# B&R Automation Studio project CombinedLinenCleanA6
Automation Studio 4.10.2.37; technology packages: mappView 5.17.0

## Configuration CP1584

CPU 5APC2200.AL14-000, AutomationRuntime B4.63, Build 4.1.2, Safety 0.0, Vc V4.72.3

### Task classes (Cpu.sw)
```
Cyclic#2 (cycle 10000 us, tolerance 10000 us):
  zzstd <- Sequences.zzstd.prg
  zztc2str <- Sequences.zztc2str.prg
  zzforcei <- Sequences.zzforcei.prg
  zzconst <- Sequences.zzconst.prg
  zztrip <- Sequences.zztrip.prg
  zzbagsfl <- Sequences.zzbagsfl.prg
  zzbitcal <- Sequences.zzbitcal.prg
  zcusfifo <- Sequences.zcusfifo.prg
  zzStnSer <- Sequences.10ms.zzStnSer.prg
  1_clu_1 <- Sequences.10ms.1_clu_1.prg
  2_cvc1 <- Sequences.10ms.2_cvc1.prg
  3_cic1 <- Sequences.10ms.3_cic1.prg
  4_cic2 <- Sequences.10ms.4_cic2.prg
  5_cic3 <- Sequences.10ms.5_cic3.prg
  6_sdc1 <- Sequences.10ms.6_sdc1.prg [disabled]
  7_sdc2 <- Sequences.10ms.7_sdc2.prg
  8_sdc3 <- Sequences.10ms.8_sdc3.prg
  9_sdc4 <- Sequences.10ms.9_sdc4.prg
  10_sdc5 <- Sequences.10ms.10_sdc5.prg
  11_sdc6 <- Sequences.10ms.11_sdc6.prg
  12_ebag <- Sequences.10ms.12_ebag.prg
  13_fb_eb <- Sequences.10ms.13_fb_eb.prg
  14_cvc2 <- Sequences.10ms.14_cvc2.prg
  15_cdc7 <- Sequences.10ms.15_cdc7.prg
  16_cic4 <- Sequences.10ms.16_cic4.prg
  17_cp12 <- Sequences.10ms.17_cp12.prg
  18_cdc8 <- Sequences.10ms.18_cdc8.prg
  19_cp13 <- Sequences.10ms.19_cp13.prg
  20_cpc1 <- Sequences.10ms.20_cpc1.prg
  21_cic6 <- Sequences.10ms.21_cic6.prg
  22_cic7 <- Sequences.10ms.22_cic7.prg
  23_Ebag <- Sequences.10ms.23_Ebag.prg
  24_csb1 <- Sequences.10ms.24_csb1.prg
  25_cp16 <- Sequences.10ms.25_cp16.prg
  26_cic8 <- Sequences.10ms.26_cic8.prg
  27_csb2 <- Sequences.10ms.27_csb2.prg
  ssr <- Sequences.10ms.ssr.prg
  can_live <- Sequences.can_live.prg
  zzio <- Sequences.zzio.prg
  zztcpip <- Sequences.zztcpip.prg
  zzuld_3 <- Sequences.zzuld_3.prg
  zzreport <- Sequences.zzreport.prg
  zztc2end <- Sequences.zztc2end.prg
Cyclic#5:
  zzweigh <- zzweigh.prg [disabled]
  can_drv2 <- Mewa.200ms.CAN.can_drv2.prg
  zzstn_q <- Sequences.zzstn_q.prg
  zzalarms <- Sequences.zzalarms.prg
  zztime <- zztime.prg
  zztc2end1 <- zztc2end.prg
DataObjects: can_cmd <- Mewa.200ms.CAN.can_cmd.dob
Binaries: TCData, udbdef, mvLoader, sysconf, ashwd, asfw, arconfig, iomap, ashwac
Libraries: DataBackUp, AsDb, standard, runtime, FileIO, Ethernet, dvframe, DataObj, OPERATOR, CAN_Lib, AsTime, AsString, SupLib4, sys_lib, AsTCP, KGstring, Visapi, AsETH, AsBrStr, AsBrWStr, AsUSB, AsMem, AsArLog, AsUDP, brsystem, AsIODiag, AsARCfg, AsIecCon, IecCheck, arssl, zzSQL_Lib
```

### Hardware
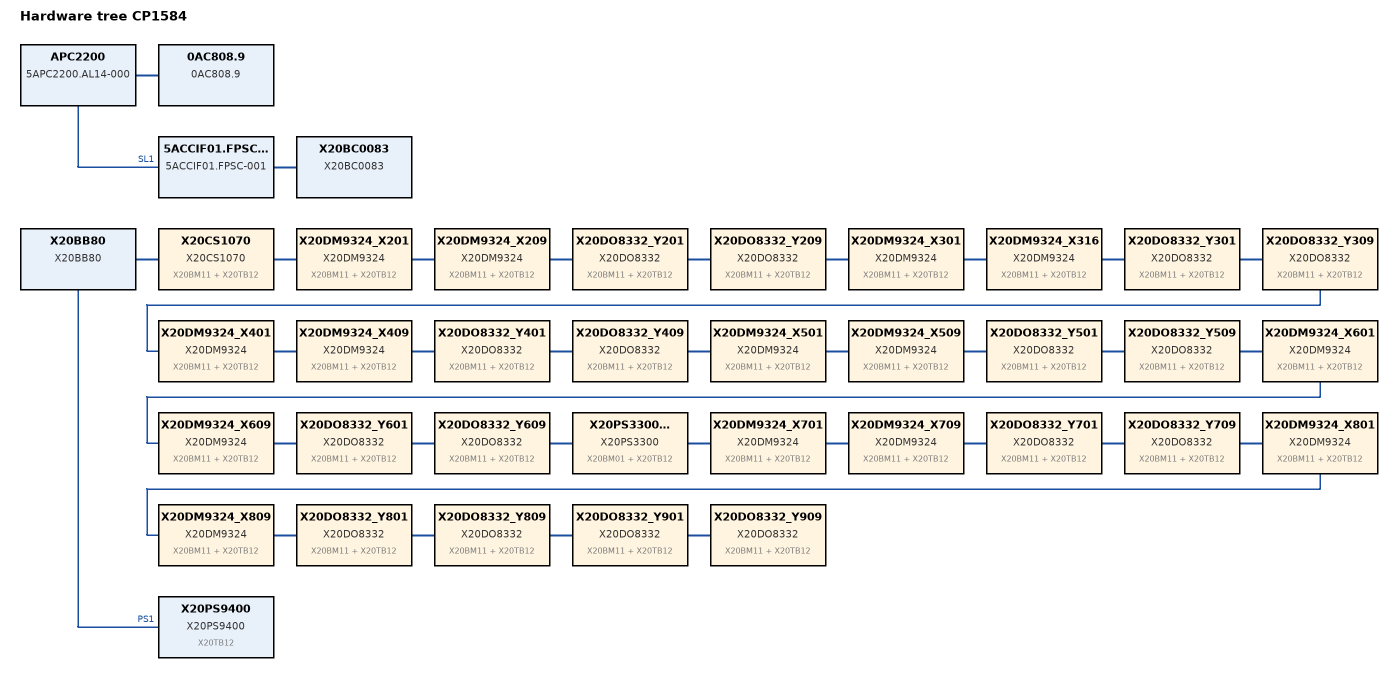
```
0AC808.9 : 0AC808.9 v1.0.0.0  [ETH1 -> APC2200.IF3 [Cable Type=PowerlinkCable, Length=10, Version=1.0.0.3]]
5ACCIF01.FPSC-001 : 5ACCIF01.FPSC-001 v1.9.1.0  [SL -> APC2200.SL1]
APC2200 : 5APC2200.AL14-000 v2.0.3.0
  Connector IF3:
    AssignedOperatingSystem = ARemb
    ActivateDevice = 1
    Baudrate = 100
    InaNodeNumber = 21
    ActivateANSL = 0
  Connector IF4:
    AssignedOperatingSystem = ARemb
    ActivateDevice = 1
    Mode = Manual
    InternetAddress = 10.8.4.21
    SubnetMask = 255.255.240.0
  Connector IF5:
    AssignedOperatingSystem = ARemb
  Connector IF6:
    AssignedOperatingSystem = ARemb
  ConfigurationID = AS4_2_BaseStandard_Supertrack
  UserRamDevice = PCI.1.PPC21xx.SRAM
  UserRamSize = 200000
  RemMemDevice = PCI.1.PPC21xx.SRAM
  RemMemSize = 200000
  PermanentPvSize = 46756
  RemanentGlobalPvSize = 8944
  VolatileGlobalPvSize = 450000
  EnableUsbRemoteInstall = 1
  EnableCfRemoteInstall = 1
  RebootPowerfail = 2
  Cyclic1Duration = 1000
  Cyclic1Tolerance = 1000
  Cyclic2Duration = 10000
  Cyclic2Tolerance = 10000
  FileDevice1
  FileDeviceName1 = USBStick
  FileDevicePath1 = /bd0\
  FileDevice2
  FileDeviceName2 = UserPart
  FileDevicePath2 = F:\
  EthernetHostName = SupertrackPLC
  EthernetDefaultGateway = 10.8.15.254
  FtpUser1
  FtpUsername1 = admin
  FtpUserPassword1 = vwQCGOhDKwuFhUdMhisKVJgiKzmoNTQazzJQnTTJsZU=  // admin
  FtpUserSalt1 = XFuy8Eo/
  FTPAccessRight1 = 0
  ActivateOpcUa = 1
  OpcUaInformationModels_PV_Version = 1
X20BB80 : X20BB80 v1.1.0.0
X20BC0083 : X20BC0083 v2.14.0.0  [PLK1 -> 5ACCIF01.FPSC-001.IF1 (NodeNumber=1) [Cable Type=PowerlinkCable, Length=10, Version=1.0.0.3]; SL -> X20BB80.SL1]
  Supervision = off
X20BM01 : X20BM01 v2.1.0.0  [X2X1 -> X20BM11t.X2X2]
X20BM11 : X20BM11 v1.1.0.0  [X2X1 -> X20BB80.IF1]
X20BM11a : X20BM11 v1.1.0.0  [X2X1 -> X20BM11.X2X2]
X20BM11aa : X20BM11 v1.1.0.0  [X2X1 -> X20BM11z.X2X2]
X20BM11ab : X20BM11 v1.1.0.0  [X2X1 -> X20BM11aa.X2X2]
X20BM11ac : X20BM11 v1.1.0.0  [X2X1 -> X20BM11ab.X2X2]
X20BM11ad : X20BM11 v1.1.0.0  [X2X1 -> X20BM11ac.X2X2]
X20BM11b : X20BM11 v1.1.0.0  [X2X1 -> X20BM11a.X2X2]
X20BM11c : X20BM11 v1.1.0.0  [X2X1 -> X20BM11b.X2X2]
X20BM11d : X20BM11 v1.1.0.0  [X2X1 -> X20BM11e.X2X2]
X20BM11e : X20BM11 v1.1.0.0  [X2X1 -> X20BM11c.X2X2]
X20BM11f : X20BM11 v1.1.0.0  [X2X1 -> X20BM11d.X2X2]
X20BM11g : X20BM11 v1.1.0.0  [X2X1 -> X20BM11s.X2X2]
X20BM11h : X20BM11 v1.1.0.0  [X2X1 -> X20BM11f.X2X2]
X20BM11i : X20BM11 v1.1.0.0  [X2X1 -> X20BM11h.X2X2]
X20BM11j : X20BM11 v1.1.0.0  [X2X1 -> X20BM11i.X2X2]
X20BM11k : X20BM11 v1.1.0.0  [X2X1 -> X20BM11j.X2X2]
X20BM11l : X20BM11 v1.1.0.0  [X2X1 -> X20BM11k.X2X2]
X20BM11m : X20BM11 v1.1.0.0  [X2X1 -> X20BM11l.X2X2]
X20BM11n : X20BM11 v1.1.0.0  [X2X1 -> X20BM11m.X2X2]
X20BM11o : X20BM11 v1.1.0.0  [X2X1 -> X20BM11n.X2X2]
X20BM11p : X20BM11 v1.1.0.0  [X2X1 -> X20BM11o.X2X2]
X20BM11q : X20BM11 v1.1.0.0  [X2X1 -> X20BM11p.X2X2]
X20BM11r : X20BM11 v1.1.0.0  [X2X1 -> X20BM11q.X2X2]
X20BM11s : X20BM11 v1.1.0.0  [X2X1 -> X20BM11r.X2X2]
X20BM11t : X20BM11 v1.1.0.0  [X2X1 -> X20BM11g.X2X2]
X20BM11u : X20BM11 v1.1.0.0  [X2X1 -> X20BM01.X2X2]
X20BM11v : X20BM11 v1.1.0.0  [X2X1 -> X20BM11u.X2X2]
X20BM11w : X20BM11 v1.1.0.0  [X2X1 -> X20BM11v.X2X2]
X20BM11x : X20BM11 v1.1.0.0  [X2X1 -> X20BM11w.X2X2]
X20BM11y : X20BM11 v1.1.0.0  [X2X1 -> X20BM11x.X2X2]
X20BM11z : X20BM11 v1.1.0.0  [X2X1 -> X20BM11y.X2X2]
X20CS1070 : X20CS1070 v1.8.0.0  [SS1 -> X20TB12af.SS; SL -> X20BM11.SL1]
  FunctionModel = Stream1xCan
  Supervision = off
X20DM9324_X201 : X20DM9324 v1.2.0.0  [SS1 -> X20TB12a.SS; SL -> X20BM11a.SL1]
  Supervision = off
X20DM9324_X209 : X20DM9324 v1.2.0.0  [SS1 -> X20TB12b.SS; SL -> X20BM11b.SL1]
  Supervision = off
X20DM9324_X301 : X20DM9324 v1.2.0.0  [SS1 -> X20TB12d.SS; SL -> X20BM11d.SL1]
  Supervision = off
X20DM9324_X316 : X20DM9324 v1.2.0.0  [SS1 -> X20TB12f.SS; SL -> X20BM11f.SL1]
  Supervision = off
X20DM9324_X401 : X20DM9324 v1.2.0.0  [SS1 -> X20TB12j.SS; SL -> X20BM11j.SL1]
  Supervision = off
X20DM9324_X409 : X20DM9324 v1.2.0.0  [SS1 -> X20TB12k.SS; SL -> X20BM11k.SL1]
  Supervision = off
X20DM9324_X501 : X20DM9324 v1.2.0.0  [SS1 -> X20TB12n.SS; SL -> X20BM11n.SL1]
  Supervision = off
X20DM9324_X509 : X20DM9324 v1.2.0.0  [SS1 -> X20TB12o.SS; SL -> X20BM11o.SL1]
  Supervision = off
X20DM9324_X601 : X20DM9324 v1.2.0.0  [SS1 -> X20TB12r.SS; SL -> X20BM11r.SL1]
  Supervision = off
X20DM9324_X609 : X20DM9324 v1.2.0.0  [SS1 -> X20TB12s.SS; SL -> X20BM11s.SL1]
  Supervision = off
X20DM9324_X701 : X20DM9324 v1.2.0.0  [SS1 -> X20TB12u.SS; SL -> X20BM11u.SL1]
  Supervision = off
X20DM9324_X709 : X20DM9324 v1.2.0.0  [SS1 -> X20TB12v.SS; SL -> X20BM11v.SL1]
  Supervision = off
X20DM9324_X801 : X20DM9324 v1.2.0.0  [SS1 -> X20TB12z.SS; SL -> X20BM11y.SL1]
  Supervision = off
X20DM9324_X809 : X20DM9324 v1.2.0.0  [SS1 -> X20TB12aa.SS; SL -> X20BM11z.SL1]
  Supervision = off
X20DO8332_Y201 : X20DO8332 v1.5.0.0  [SS1 -> X20TB12c.SS; SL -> X20BM11c.SL1]
  Supervision = off
X20DO8332_Y209 : X20DO8332 v1.5.0.0  [SS1 -> X20TB12e.SS; SL -> X20BM11e.SL1]
  Supervision = off
X20DO8332_Y301 : X20DO8332 v1.5.0.0  [SS1 -> X20TB12h.SS; SL -> X20BM11h.SL1]
  Supervision = off
X20DO8332_Y309 : X20DO8332 v1.5.0.0  [SS1 -> X20TB12i.SS; SL -> X20BM11i.SL1]
  Supervision = off
X20DO8332_Y401 : X20DO8332 v1.5.0.0  [SS1 -> X20TB12l.SS; SL -> X20BM11l.SL1]
  Supervision = off
X20DO8332_Y409 : X20DO8332 v1.5.0.0  [SS1 -> X20TB12m.SS; SL -> X20BM11m.SL1]
  Supervision = off
X20DO8332_Y501 : X20DO8332 v1.5.0.0  [SS1 -> X20TB12p.SS; SL -> X20BM11p.SL1]
  Supervision = off
X20DO8332_Y509 : X20DO8332 v1.5.0.0  [SS1 -> X20TB12q.SS; SL -> X20BM11q.SL1]
  Supervision = off
X20DO8332_Y601 : X20DO8332 v1.5.0.0  [SS1 -> X20TB12g.SS; SL -> X20BM11g.SL1]
  Supervision = off
X20DO8332_Y609 : X20DO8332 v1.5.0.0  [SS1 -> X20TB12t.SS; SL -> X20BM11t.SL1]
  Supervision = off
X20DO8332_Y701 : X20DO8332 v1.5.0.0  [SS1 -> X20TB12x.SS; SL -> X20BM11w.SL1]
  Supervision = off
X20DO8332_Y709 : X20DO8332 v1.5.0.0  [SS1 -> X20TB12y.SS; SL -> X20BM11x.SL1]
  Supervision = off
X20DO8332_Y801 : X20DO8332 v1.5.0.0  [SS1 -> X20TB12ab.SS; SL -> X20BM11aa.SL1]
  Supervision = off
X20DO8332_Y809 : X20DO8332 v1.5.0.0  [SS1 -> X20TB12ac.SS; SL -> X20BM11ab.SL1]
  Supervision = off
X20DO8332_Y901 : X20DO8332 v1.5.0.0  [SS1 -> X20TB12ad.SS; SL -> X20BM11ac.SL1]
  Supervision = off
X20DO8332_Y909 : X20DO8332 v1.5.0.0  [SS1 -> X20TB12ae.SS; SL -> X20BM11ad.SL1]
  Supervision = off
X20PS3300_Power : X20PS3300 v1.3.0.0  [SS1 -> X20TB12w.SS; SL -> X20BM01.SL1]
  Supervision = off
X20PS9400 : X20PS9400 v1.8.0.0  [SS1 -> X20TB12.SS; PS -> X20BB80.PS1]
  Supervision = off
X20TB12 : X20TB12 v1.0.0.0
X20TB12a : X20TB12 v1.0.0.0
X20TB12aa : X20TB12 v1.0.0.0
X20TB12ab : X20TB12 v1.0.0.0
X20TB12ac : X20TB12 v1.0.0.0
X20TB12ad : X20TB12 v1.0.0.0
X20TB12ae : X20TB12 v1.0.0.0
X20TB12af : X20TB12 v1.0.0.0
X20TB12b : X20TB12 v1.0.0.0
X20TB12c : X20TB12 v1.0.0.0
X20TB12d : X20TB12 v1.0.0.0
X20TB12e : X20TB12 v1.0.0.0
X20TB12f : X20TB12 v1.0.0.0
X20TB12g : X20TB12 v1.0.0.0
X20TB12h : X20TB12 v1.0.0.0
X20TB12i : X20TB12 v1.0.0.0
X20TB12j : X20TB12 v1.0.0.0
X20TB12k : X20TB12 v1.0.0.0
X20TB12l : X20TB12 v1.0.0.0
X20TB12m : X20TB12 v1.0.0.0
X20TB12n : X20TB12 v1.0.0.0
X20TB12o : X20TB12 v1.0.0.0
X20TB12p : X20TB12 v1.0.0.0
X20TB12q : X20TB12 v1.0.0.0
X20TB12r : X20TB12 v1.0.0.0
X20TB12s : X20TB12 v1.0.0.0
X20TB12t : X20TB12 v1.0.0.0
X20TB12u : X20TB12 v1.0.0.0
X20TB12v : X20TB12 v1.0.0.0
X20TB12w : X20TB12 v1.0.0.0
X20TB12x : X20TB12 v1.0.0.0
X20TB12y : X20TB12 v1.0.0.0
X20TB12z : X20TB12 v1.0.0.0
```

### IoMap.iom - APC2200/IoMap.iom
```iecst
(********************************************************************
 * COPYRIGHT --
 ********************************************************************
 * File: IoMap.iom
 * Author: Dave
 * Created: November 19, 2010
 ********************************************************************
 * IO mapping file
 ********************************************************************)
VAR_CONFIG
	X[2].X01 AT %IX."X20DM9324_X201".DigitalInput01;
	X[2].X02 AT %IX."X20DM9324_X201".DigitalInput02;
	X[2].X03 AT %IX."X20DM9324_X201".DigitalInput03;
	X[2].X04 AT %IX."X20DM9324_X201".DigitalInput04;
	X[2].X05 AT %IX."X20DM9324_X201".DigitalInput05;
	X[2].X06 AT %IX."X20DM9324_X201".DigitalInput06;
	X[2].X07 AT %IX."X20DM9324_X201".DigitalInput07;
	X[2].X08 AT %IX."X20DM9324_X201".DigitalInput08;
	X[2].X09 AT %IX."X20DM9324_X209".DigitalInput01;
	X[2].X10 AT %IX."X20DM9324_X209".DigitalInput02;
	X[2].X11 AT %IX."X20DM9324_X209".DigitalInput03;
	X[2].X12 AT %IX."X20DM9324_X209".DigitalInput04;
	X[2].X13 AT %IX."X20DM9324_X209".DigitalInput05;
	X[2].X14 AT %IX."X20DM9324_X209".DigitalInput06;
	X[2].X15 AT %IX."X20DM9324_X209".DigitalInput07;
	X[2].X16 AT %IX."X20DM9324_X209".DigitalInput08;
	Y[2].Y01 AT %QX."X20DO8332_Y201".DigitalOutput01;
	Y[2].Y02 AT %QX."X20DO8332_Y201".DigitalOutput02;
	Y[2].Y03 AT %QX."X20DO8332_Y201".DigitalOutput03;
	Y[2].Y04 AT %QX."X20DO8332_Y201".DigitalOutput04;
	Y[2].Y05 AT %QX."X20DO8332_Y201".DigitalOutput05;
	Y[2].Y06 AT %QX."X20DO8332_Y201".DigitalOutput06;
	Y[2].Y07 AT %QX."X20DO8332_Y201".DigitalOutput07;
	Y[2].Y08 AT %QX."X20DO8332_Y201".DigitalOutput08;
	Y[2].Y09 AT %QX."X20DO8332_Y209".DigitalOutput01;
	Y[2].Y10 AT %QX."X20DO8332_Y209".DigitalOutput02;
	Y[2].Y11 AT %QX."X20DO8332_Y209".DigitalOutput03;
	Y[2].Y12 AT %QX."X20DO8332_Y209".DigitalOutput04;
	Y[2].Y13 AT %QX."X20DO8332_Y209".DigitalOutput05;
	Y[2].Y14 AT %QX."X20DO8332_Y209".DigitalOutput06;
	Y[2].Y15 AT %QX."X20DO8332_Y209".DigitalOutput07;
	Y[2].Y16 AT %QX."X20DO8332_Y209".DigitalOutput08;
	X[3].X01 AT %IX."X20DM9324_X301".DigitalInput01;
	X[3].X02 AT %IX."X20DM9324_X301".DigitalInput02;
	X[3].X03 AT %IX."X20DM9324_X301".DigitalInput03;
	X[3].X04 AT %IX."X20DM9324_X301".DigitalInput04;
	X[3].X05 AT %IX."X20DM9324_X301".DigitalInput05;
	X[3].X06 AT %IX."X20DM9324_X301".DigitalInput06;
	X[3].X07 AT %IX."X20DM9324_X301".DigitalInput07;
	X[3].X08 AT %IX."X20DM9324_X301".DigitalInput08;
	X[3].X09 AT %IX."X20DM9324_X316".DigitalInput01;
	X[3].X10 AT %IX."X20DM9324_X316".DigitalInput02;
	X[3].X11 AT %IX."X20DM9324_X316".DigitalInput03;
	X[3].X12 AT %IX."X20DM9324_X316".DigitalInput04;
	X[3].X13 AT %IX."X20DM9324_X316".DigitalInput05;
	X[3].X14 AT %IX."X20DM9324_X316".DigitalInput06;
	X[3].X15 AT %IX."X20DM9324_X316".DigitalInput07;
	X[3].X16 AT %IX."X20DM9324_X316".DigitalInput08;
	Y[3].Y01 AT %QX."X20DO8332_Y301".DigitalOutput01;
	Y[3].Y02 AT %QX."X20DO8332_Y301".DigitalOutput02;
	Y[3].Y03 AT %QX."X20DO8332_Y301".DigitalOutput03;
	Y[3].Y04 AT %QX."X20DO8332_Y301".DigitalOutput04;
	Y[3].Y05 AT %QX."X20DO8332_Y301".DigitalOutput05;
	Y[3].Y06 AT %QX."X20DO8332_Y301".DigitalOutput06;
	Y[3].Y07 AT %QX."X20DO8332_Y301".DigitalOutput07;
	Y[3].Y08 AT %QX."X20DO8332_Y301".DigitalOutput08;
	Y[3].Y09 AT %QX."X20DO8332_Y309".DigitalOutput01;
	Y[3].Y10 AT %QX."X20DO8332_Y309".DigitalOutput02;
	Y[3].Y11 AT %QX."X20DO8332_Y309".DigitalOutput03;
	Y[3].Y12 AT %QX."X20DO8332_Y309".DigitalOutput04;
	Y[3].Y13 AT %QX."X20DO8332_Y309".DigitalOutput05;
	Y[3].Y14 AT %QX."X20DO8332_Y309".DigitalOutput06;
	Y[3].Y15 AT %QX."X20DO8332_Y309".DigitalOutput07;
	Y[3].Y16 AT %QX."X20DO8332_Y309".DigitalOutput08;
	X[4].X01 AT %IX."X20DM9324_X401".DigitalInput01;
	X[4].X02 AT %IX."X20DM9324_X401".DigitalInput02;
	X[4].X03 AT %IX."X20DM9324_X401".DigitalInput03;
	X[4].X04 AT %IX."X20DM9324_X401".DigitalInput04;
	X[4].X05 AT %IX."X20DM9324_X401".DigitalInput05;
	X[4].X06 AT %IX."X20DM9324_X401".DigitalInput06;
	X[4].X07 AT %IX."X20DM9324_X401".DigitalInput07;
	X[4].X08 AT %IX."X20DM9324_X401".DigitalInput08;
	X[4].X09 AT %IX."X20DM9324_X409".DigitalInput01;
	X[4].X10 AT %IX."X20DM9324_X409".DigitalInput02;
	X[4].X11 AT %IX."X20DM9324_X409".DigitalInput03;
	X[4].X12 AT %IX."X20DM9324_X409".DigitalInput04;
	X[4].X13 AT %IX."X20DM9324_X409".DigitalInput05;
	X[4].X14 AT %IX."X20DM9324_X409".DigitalInput06;
	X[4].X15 AT %IX."X20DM9324_X409".DigitalInput07;
	X[4].X16 AT %IX."X20DM9324_X409".DigitalInput08;
	Y[4].Y01 AT %QX."X20DO8332_Y401".DigitalOutput01;
	Y[4].Y02 AT %QX."X20DO8332_Y401".DigitalOutput02;
	Y[4].Y03 AT %QX."X20DO8332_Y401".DigitalOutput03;
	Y[4].Y04 AT %QX."X20DO8332_Y401".DigitalOutput04;
	Y[4].Y05 AT %QX."X20DO8332_Y401".DigitalOutput05;
	Y[4].Y06 AT %QX."X20DO8332_Y401".DigitalOutput06;
	Y[4].Y07 AT %QX."X20DO8332_Y401".DigitalOutput07;
	Y[4].Y08 AT %QX."X20DO8332_Y401".DigitalOutput08;
	Y[4].Y09 AT %QX."X20DO8332_Y409".DigitalOutput01;
	Y[4].Y10 AT %QX."X20DO8332_Y409".DigitalOutput02;
	Y[4].Y11 AT %QX."X20DO8332_Y409".DigitalOutput03;
	Y[4].Y12 AT %QX."X20DO8332_Y409".DigitalOutput04;
	Y[4].Y13 AT %QX."X20DO8332_Y409".DigitalOutput05;
	Y[4].Y14 AT %QX."X20DO8332_Y409".DigitalOutput06;
	Y[4].Y15 AT %QX."X20DO8332_Y409".DigitalOutput07;
	Y[4].Y16 AT %QX."X20DO8332_Y409".DigitalOutput08;
	X[5].X01 AT %IX."X20DM9324_X501".DigitalInput01;
	X[5].X02 AT %IX."X20DM9324_X501".DigitalInput02;
	X[5].X03 AT %IX."X20DM9324_X501".DigitalInput03;
	X[5].X04 AT %IX."X20DM9324_X501".DigitalInput04;
	X[5].X05 AT %IX."X20DM9324_X501".DigitalInput05;
	X[5].X06 AT %IX."X20DM9324_X501".DigitalInput06;
	X[5].X07 AT %IX."X20DM9324_X501".DigitalInput07;
	X[5].X08 AT %IX."X20DM9324_X501".DigitalInput08;
	X[5].X09 AT %IX."X20DM9324_X509".DigitalInput01;
	X[5].X10 AT %IX."X20DM9324_X509".DigitalInput02;
	X[5].X11 AT %IX."X20DM9324_X509".DigitalInput03;
	X[5].X12 AT %IX."X20DM9324_X509".DigitalInput04;
	X[5].X13 AT %IX."X20DM9324_X509".DigitalInput05;
	X[5].X14 AT %IX."X20DM9324_X509".DigitalInput06;
	X[5].X15 AT %IX."X20DM9324_X509".DigitalInput07;
	X[5].X16 AT %IX."X20DM9324_X509".DigitalInput08;
	Y[5].Y01 AT %QX."X20DO8332_Y501".DigitalOutput01;
	Y[5].Y02 AT %QX."X20DO8332_Y501".DigitalOutput02;
	Y[5].Y03 AT %QX."X20DO8332_Y501".DigitalOutput03;
	Y[5].Y04 AT %QX."X20DO8332_Y501".DigitalOutput04;
	Y[5].Y05 AT %QX."X20DO8332_Y501".DigitalOutput05;
	Y[5].Y06 AT %QX."X20DO8332_Y501".DigitalOutput06;
	Y[5].Y07 AT %QX."X20DO8332_Y501".DigitalOutput07;
	Y[5].Y08 AT %QX."X20DO8332_Y501".DigitalOutput08;
	Y[5].Y09 AT %QX."X20DO8332_Y509".DigitalOutput01;
	Y[5].Y10 AT %QX."X20DO8332_Y509".DigitalOutput02;
	Y[5].Y11 AT %QX."X20DO8332_Y509".DigitalOutput03;
	Y[5].Y12 AT %QX."X20DO8332_Y509".DigitalOutput04;
	Y[5].Y13 AT %QX."X20DO8332_Y509".DigitalOutput05;
	Y[5].Y14 AT %QX."X20DO8332_Y509".DigitalOutput06;
	Y[5].Y15 AT %QX."X20DO8332_Y509".DigitalOutput07;
	Y[5].Y16 AT %QX."X20DO8332_Y509".DigitalOutput08;
	X[6].X01 AT %IX."X20DM9324_X601".DigitalInput01;
	X[6].X02 AT %IX."X20DM9324_X601".DigitalInput02;
	X[6].X03 AT %IX."X20DM9324_X601".DigitalInput03;
	X[6].X04 AT %IX."X20DM9324_X601".DigitalInput04;
	X[6].X05 AT %IX."X20DM9324_X601".DigitalInput05;
	X[6].X06 AT %IX."X20DM9324_X601".DigitalInput06;
	X[6].X07 AT %IX."X20DM9324_X601".DigitalInput07;
	X[6].X08 AT %IX."X20DM9324_X601".DigitalInput08;
	X[6].X09 AT %IX."X20DM9324_X609".DigitalInput01;
	X[6].X10 AT %IX."X20DM9324_X609".DigitalInput02;
	X[6].X11 AT %IX."X20DM9324_X609".DigitalInput03;
	X[6].X12 AT %IX."X20DM9324_X609".DigitalInput04;
	X[6].X13 AT %IX."X20DM9324_X609".DigitalInput05;
	X[6].X14 AT %IX."X20DM9324_X609".DigitalInput06;
	X[6].X15 AT %IX."X20DM9324_X609".DigitalInput07;
	X[6].X16 AT %IX."X20DM9324_X609".DigitalInput08;
	Y[6].Y01 AT %QX."X20DO8332_Y601".DigitalOutput01;
	Y[6].Y02 AT %QX."X20DO8332_Y601".DigitalOutput02;
	Y[6].Y03 AT %QX."X20DO8332_Y601".DigitalOutput03;
	Y[6].Y04 AT %QX."X20DO8332_Y601".DigitalOutput04;
	Y[6].Y05 AT %QX."X20DO8332_Y601".DigitalOutput05;
	Y[6].Y06 AT %QX."X20DO8332_Y601".DigitalOutput06;
	Y[6].Y07 AT %QX."X20DO8332_Y601".DigitalOutput07;
	Y[6].Y08 AT %QX."X20DO8332_Y601".DigitalOutput08;
	Y[6].Y09 AT %QX."X20DO8332_Y609".DigitalOutput01;
	Y[6].Y10 AT %QX."X20DO8332_Y609".DigitalOutput02;
	Y[6].Y11 AT %QX."X20DO8332_Y609".DigitalOutput03;
	Y[6].Y12 AT %QX."X20DO8332_Y609".DigitalOutput04;
	Y[6].Y13 AT %QX."X20DO8332_Y609".DigitalOutput05;
	Y[6].Y14 AT %QX."X20DO8332_Y609".DigitalOutput06;
	Y[6].Y15 AT %QX."X20DO8332_Y609".DigitalOutput07;
	Y[6].Y16 AT %QX."X20DO8332_Y609".DigitalOutput08;
	X[7].X01 AT %IX."X20DM9324_X701".DigitalInput01;
	X[7].X02 AT %IX."X20DM9324_X701".DigitalInput02;
	X[7].X03 AT %IX."X20DM9324_X701".DigitalInput03;
	X[7].X04 AT %IX."X20DM9324_X701".DigitalInput04;
	X[7].X05 AT %IX."X20DM9324_X701".DigitalInput05;
	X[7].X06 AT %IX."X20DM9324_X701".DigitalInput06;
	X[7].X07 AT %IX."X20DM9324_X701".DigitalInput07;
	X[7].X08 AT %IX."X20DM9324_X701".DigitalInput08;
	X[7].X09 AT %IX."X20DM9324_X709".DigitalInput01;
	X[7].X10 AT %IX."X20DM9324_X709".DigitalInput02;
	X[7].X11 AT %IX."X20DM9324_X709".DigitalInput03;
	X[7].X12 AT %IX."X20DM9324_X709".DigitalInput04;
	X[7].X13 AT %IX."X20DM9324_X709".DigitalInput05;
	X[7].X14 AT %IX."X20DM9324_X709".DigitalInput06;
	X[7].X15 AT %IX."X20DM9324_X709".DigitalInput07;
	X[7].X16 AT %IX."X20DM9324_X709".DigitalInput08;
	Y[7].Y01 AT %QX."X20DO8332_Y701".DigitalOutput01;
	Y[7].Y02 AT %QX."X20DO8332_Y701".DigitalOutput02;
	Y[7].Y03 AT %QX."X20DO8332_Y701".DigitalOutput03;
	Y[7].Y04 AT %QX."X20DO8332_Y701".DigitalOutput04;
	Y[7].Y05 AT %QX."X20DO8332_Y701".DigitalOutput05;
	Y[7].Y06 AT %QX."X20DO8332_Y701".DigitalOutput06;
	Y[7].Y07 AT %QX."X20DO8332_Y701".DigitalOutput07;
	Y[7].Y08 AT %QX."X20DO8332_Y701".DigitalOutput08;
	Y[7].Y09  AT %QX."X20DO8332_Y709".DigitalOutput01;
	Y[7].Y10  AT %QX."X20DO8332_Y709".DigitalOutput02;
	Y[7].Y11  AT %QX."X20DO8332_Y709".DigitalOutput03;
	Y[7].Y12  AT %QX."X20DO8332_Y709".DigitalOutput04;
	Y[7].Y13  AT %QX."X20DO8332_Y709".DigitalOutput05;
	Y[7].Y14  AT %QX."X20DO8332_Y709".DigitalOutput06;
	Y[7].Y15  AT %QX."X20DO8332_Y709".DigitalOutput07;
	Y[7].Y16  AT %QX."X20DO8332_Y709".DigitalOutput08;
	X[8].X01 AT %IX."X20DM9324_X801".DigitalInput01;
	X[8].X02  AT %IX."X20DM9324_X801".DigitalInput02;
	X[8].X03  AT %IX."X20DM9324_X801".DigitalInput03;
	X[8].X04  AT %IX."X20DM9324_X801".DigitalInput04;
	X[8].X05  AT %IX."X20DM9324_X801".DigitalInput05;
	X[8].X06  AT %IX."X20DM9324_X801".DigitalInput06;
	X[8].X07  AT %IX."X20DM9324_X801".DigitalInput07;
	X[8].X08  AT %IX."X20DM9324_X801".DigitalInput08;
	X[8].X09  AT %IX."X20DM9324_X809".DigitalInput01;
	X[8].X10  AT %IX."X20DM9324_X809".DigitalInput02;
	X[8].X11  AT %IX."X20DM9324_X809".DigitalInput03;
	X[8].X12  AT %IX."X20DM9324_X809".DigitalInput04;
	X[8].X13  AT %IX."X20DM9324_X809".DigitalInput05;
	X[8].X14  AT %IX."X20DM9324_X809".DigitalInput06;
	X[8].X15  AT %IX."X20DM9324_X809".DigitalInput07;
	X[8].X16  AT %IX."X20DM9324_X809".DigitalInput08;
	Y[8].Y01 AT %QX."X20DO8332_Y801".DigitalOutput01;
	Y[8].Y02  AT %QX."X20DO8332_Y801".DigitalOutput02;
	Y[8].Y03  AT %QX."X20DO8332_Y801".DigitalOutput03;
	Y[8].Y04  AT %QX."X20DO8332_Y801".DigitalOutput04;
	Y[8].Y05  AT %QX."X20DO8332_Y801".DigitalOutput05;
	Y[8].Y06  AT %QX."X20DO8332_Y801".DigitalOutput06;
	Y[8].Y07  AT %QX."X20DO8332_Y801".DigitalOutput07;
	Y[8].Y08  AT %QX."X20DO8332_Y801".DigitalOutput08;
	Y[8].Y09  AT %QX."X20DO8332_Y809".DigitalOutput01;
	Y[8].Y10  AT %QX."X20DO8332_Y809".DigitalOutput02;
	Y[8].Y11  AT %QX."X20DO8332_Y809".DigitalOutput03;
	Y[8].Y12  AT %QX."X20DO8332_Y809".DigitalOutput04;
	Y[8].Y13  AT %QX."X20DO8332_Y809".DigitalOutput05;
	Y[8].Y14  AT %QX."X20DO8332_Y809".DigitalOutput06;
	Y[8].Y15  AT %QX."X20DO8332_Y809".DigitalOutput07;
	Y[8].Y16  AT %QX."X20DO8332_Y809".DigitalOutput08;
	Y[9].Y01 AT %QX."X20DO8332_Y901".DigitalOutput01;
	Y[9].Y02  AT %QX."X20DO8332_Y901".DigitalOutput02;
	Y[9].Y03  AT %QX."X20DO8332_Y901".DigitalOutput03;
	Y[9].Y04  AT %QX."X20DO8332_Y901".DigitalOutput04;
	Y[9].Y05  AT %QX."X20DO8332_Y901".DigitalOutput05;
	Y[9].Y06  AT %QX."X20DO8332_Y901".DigitalOutput06;
	Y[9].Y07  AT %QX."X20DO8332_Y901".DigitalOutput07;
	Y[9].Y08  AT %QX."X20DO8332_Y901".DigitalOutput08;
	Y[9].Y09  AT %QX."X20DO8332_Y909".DigitalOutput01;
	Y[9].Y10  AT %QX."X20DO8332_Y909".DigitalOutput02;
	Y[9].Y11  AT %QX."X20DO8332_Y909".DigitalOutput03;
	Y[9].Y12  AT %QX."X20DO8332_Y909".DigitalOutput04;
	Y[9].Y13  AT %QX."X20DO8332_Y909".DigitalOutput05;
	Y[9].Y14  AT %QX."X20DO8332_Y909".DigitalOutput06;
	Y[9].Y15  AT %QX."X20DO8332_Y909".DigitalOutput07;
	Y[9].Y16  AT %QX."X20DO8332_Y909".DigitalOutput08;
END_VAR
```

## Configuration DisplayPCT04

### Cpu.per - PCT04/Cpu.per
```iecst
(********************************************************************
 * COPYRIGHT -- HP
 ********************************************************************
 * File: Cpu.per
 * Author: treamsbottom
 * Created: February 28, 2012
 ********************************************************************
 * Declaration of permanent variables
 ********************************************************************)
VAR_CONFIG
	ClientServerIP AT %M0; (* *)
END_VAR
```

## Configuration Supertrack

CPU , AutomationRuntime C4.72, Build 4.1.2, Safety 1.10, Vc V4.72.0

## Logical view

Binary libraries used (declarations not repeated): standard, runtime, FileIO, Ethernet, dvframe, DataObj, OPERATOR, AsTime, AsString, AsCANopen, sys_lib, AsTCP, KGstring, CAN_Lib, Visapi, AsARCfg, AsETH, AsDb, brsystem, AsUSB, AsMem, AsArLog, AsBrWStr, AsUDP, AsIODiag, AsBrStr, AsIecCon, IecCheck, DataBackUp

### Program Logical/Reference/4_ppn1 (IEC) - *ppn

#### ppn.var
```iecst
VAR RETAIN
	LASTSTEP : UINT;
	PLS : BOOL;
	STEP : UINT;
END_VAR
VAR
	TimerAlarm : TON_10ms;
	mySeq : UINT;
	myIO : UINT;
	I_BagAtSep : ARRAY[0..3] OF BOOL;
	I_BagInSep : ARRAY[0..3] OF BOOL;
	O_SelectLine : ARRAY[0..3] OF BOOL;
	O_SelectDest : ARRAY[0..30] OF BOOL;
	TON_Settled : ARRAY[0..3] OF TON_10ms;
	n : UINT;
	myBag : UINT;
	myBuffBag : ARRAY[0..3] OF UINT;
	LineValid : ARRAY[0..30] OF BOOL;
	myRelLine : UINT;
END_VAR
VAR RETAIN
	CurrentDest : UINT;
	CurrentLine : UINT;
END_VAR
VAR
	myDestBag : UINT;
	LineBatchCount : ARRAY[0..3] OF UINT;
	MaxBatchSize : UINT;
	ResetRequired : BOOL;
	ResetPoints : BOOL;
	ResetPointsET : UDINT;
	PrevDest : UINT;
	PrevLine : UINT;
	O_OpenSep : ARRAY[0..3] OF BOOL;
	Released : BOOL;
	myDestLine : UINT;
	ReleaseValid : BOOL;
	ClearCounts : BOOL;
	LineSearchCount : UINT;
	DestSearchCount : UINT;
	ScanUpdate : BOOL;
	ScanUpdateET : UDINT;
	MaxLines : UINT;
	LineSelect : ARRAY[0..29] OF BOOL;
	LineReset : ARRAY[0..29] OF BOOL;
	myZone : INT;
	I_BagReleased : BOOL;
	TON_BagInSep : ARRAY[0..3] OF TON_10ms;
	BufferBag : UINT;
	StorageLineLastBag : UINT;
	DebugCount : UDINT;
END_VAR
```

### Program Logical/Reference/6_pwb1 (IEC) - *PWB1 Weigh beam 1

#### pwb.ab
```automation-basic
;--------------------------------------------
;Sequence 0 - XXX0  D[900 + mySeq]
;--------------------------------------------

PROGRAM _INIT
(* init program *)
END_PROGRAM

PROGRAM _CYCLIC

;Inputs
mySeq				= 6	;Sequence number
myIO				= 343
myBag				= 776
myRelLine			= 62
myLP				= 1
myDisplayBag		= myBag
myZone				= 3

myOutBag			= Line[myRelLine].LastBag

SettleTime			= 300

I_BagInBeam			= X[myIO].X02

O_OpenSep			= FALSE

EnableRel.LP[myLP]	= FALSE

Alarm[mySeq].Name 	= 0
Alarm[mySeq].Bag	= myBag
Alarm[mySeq].Beacon	= TRUE
Alarm[mySeq].Extra	= 0
Alarm[mySeq].Time	= 3000

RawWgt = DINT(AI1223Raw[myLP])
RawWgt = (RawWgt * 2000)
IF (RawWgt > 0) THEN
	Wgt = INT(RawWgt / 32767)
ELSE
	Wgt = 0
ENDIF
IF (myBag <> myDisplayBag) THEN
	Bag[myDisplayBag].Cat = 1
	Bag[myDisplayBag].Wgt = Wgt
ENDIF

;Setup Sequence
STEP = D[900 + mySeq]
;Setup Pulse contact
PLS = (STEP <> LASTSTEP)
LASTSTEP = STEP

;Sequence
IF (STEP = 0) THEN
	;Disabled
ENDIF
WeighBeamClear = (Bag[myBag].Cat = 0) AND NOT I_BagInBeam

;Step 1 Check Weigh beam is clear
IF (STEP = 1) THEN
		IF (WeighBeamClear AND NOT Std.HaltSysZone[myZone])  THEN
		D[900 + mySeq]  = 2
	ELSE IF (Bag[myBag].Cat > 0) THEN
		Alarm[mySeq].Name = almBagDataError
	ELSE IF I_BagInBeam THEN
		Alarm[mySeq].Name = almSwitchFault
	ENDIF
ENDIF

;Step 2 Enable Release from Loading point
IF (STEP = 2) THEN
	EnableRel.LP[myLP] = WeighBeamClear
	IF I_BagInBeam AND (Bag[myBag].Cat > 0) THEN
		D[900 + mySeq] = 3
	ELSE IF (Bag[myBag].Cat > 0) THEN
		Alarm[mySeq].Name = almBagDataError
	ELSE IF I_BagInBeam THEN
		Alarm[mySeq].Name = almSwitchFault
	ENDIF
ENDIF

;Step 3 bag settles in weigh beam
TON_10ms(I_BagInBeam,SettleTime,BagSettled,BagSettledET)
IF (STEP = 3) THEN
	IF BagSettled AND (Bag[myBag].Cat > 0) AND (ReportLoading[myLP].Cat = 0) THEN
		Bag[myBag].Wgt = Wgt/10

		ReportLoading[myLP].Prg = Bag[myBag].Prg 			;Program
		ReportLoading[myLP].Cat = Bag[myBag].Cat			;Category
		ReportLoading[myLP].Cus = Bag[myBag].Cus			;Customer
		ReportLoading[myLP].Wgt = Bag[myBag].Wgt			;Weight
		ReportLoading[myLP].Cnt = 0							;Count
		ReportLoading[myLP].Stn = myLP         			;Station
		ReportLoading[myLP].Mcn = 0						;Machine
		ReportLoading[myLP].Bid = Bag[myBag].Bid			;Batch ID
		D[900 + mySeq] = 4
	ELSE IF NOT BagSettled THEN
		Alarm[mySeq].Name = almBagNotSettled
	ELSE IF (Bag[myBag].Cat = 0) THEN
		Alarm[mySeq].Name = almBagDataError
	ELSE IF (ReportLoading[myLP].Cat > 0) THEN
		Alarm[mySeq].Name = almGeneralSequence
	ENDIF
ENDIF

OkToRelease = (Bag[myBag].Cat > 0) AND Line[myRelLine].Clear  AND NOT Line[myRelLine].TripFault
;Step 4 Check for line space
IF (STEP = 4) THEN
	IF OkToRelease THEN
		D[900 + mySeq]  = 5
	ELSE IF (Bag[myBag].Cat = 0) THEN
		Alarm[mySeq].Name = almBagDataError
	ELSE IF Line[myRelLine].TripFault THEN
		Alarm[mySeq].Name = almSwitchFault
	ENDIF
ENDIF

;Step 5 Release Bag
IF (STEP = 5) THEN
	O_OpenSep = OkToRelease
	IF Line[myRelLine].Trip THEN
		Bag[myOutBag] = Bag[myBag]
		Bag[myBag] = Bag[0]
		D[900 + mySeq] = 1
	ENDIF
	IF (Bag[myBag].Cat = 0) THEN
		Alarm[mySeq].Name = almBagDataError
	ELSE IF Line[myRelLine].TripFault THEN
		Alarm[mySeq].Name = almSwitchFault
	ENDIF
ENDIF

;-----------------------------------
;PLC Outputs - adjust to suit system
;-----------------------------------

Y[myIO].Y05 = O_OpenSep

;Alarms
TimerAlarm.IN 		= NOT PLS AND (Alarm[mySeq].Name > 0)
TimerAlarm.PT 		= Alarm[mySeq].Time
TimerAlarm FUB TON_10ms()
Alarm[mySeq].On 	= TimerAlarm.Q
Alarm[mySeq].ET 	= TimerAlarm.ET
Alarm[mySeq].Zone 	= myZone
END_PROGRAM
```

### Program Logical/Reference/7_pwb2 (IEC) - *PWB2 Weigh beam 2

#### pwb.ab
```automation-basic
;--------------------------------------------
;Sequence 0 - XXX0  D[900 + mySeq]
;--------------------------------------------

PROGRAM _INIT
(* init program *)
END_PROGRAM

PROGRAM _CYCLIC

;Inputs
mySeq				= 7	;Sequence number
myIO				= 341
myBag				= 781
myRelLine			= 61
myLP				= 2
myDisplayBag		= myBag
myZone				= 3

myOutBag			= Line[myRelLine].LastBag

SettleTime			= 300

I_BagInBeam			= X[myIO].X02

O_OpenSep			= FALSE

EnableRel.LP[myLP]	= FALSE

Alarm[mySeq].Name 	= 0
Alarm[mySeq].Bag	= myBag
Alarm[mySeq].Beacon	= TRUE
Alarm[mySeq].Extra	= 0
Alarm[mySeq].Time	= 3000

RawWgt = DINT(AI1223Raw[myLP])
RawWgt = (RawWgt * 2000)
IF (RawWgt > 0) THEN
	Wgt = INT(RawWgt / 32767)
ELSE
	Wgt = 0
ENDIF
IF (myBag <> myDisplayBag) THEN
	Bag[myDisplayBag].Cat = 1
	Bag[myDisplayBag].Wgt = Wgt
ENDIF

;Setup Sequence
STEP = D[900 + mySeq]
;Setup Pulse contact
PLS = (STEP <> LASTSTEP)
LASTSTEP = STEP

;Sequence
IF (STEP = 0) THEN
	;Disabled
ENDIF
WeighBeamClear = (Bag[myBag].Cat = 0) AND NOT I_BagInBeam

;Step 1 Check Weigh beam is clear
IF (STEP = 1) THEN
	IF (WeighBeamClear AND NOT Std.HaltSysZone[myZone])  THEN
		D[900 + mySeq]  = 2
	ELSE IF (Bag[myBag].Cat > 0) THEN
		Alarm[mySeq].Name = almBagDataError
	ELSE IF I_BagInBeam THEN
		Alarm[mySeq].Name = almSwitchFault
	ENDIF
ENDIF

;Step 2 Enable Release from Loading point
IF (STEP = 2) THEN
	EnableRel.LP[myLP] = WeighBeamClear
	IF I_BagInBeam AND (Bag[myBag].Cat > 0) THEN
		D[900 + mySeq] = 3
	ELSE IF (Bag[myBag].Cat > 0) THEN
		Alarm[mySeq].Name = almBagDataError
	ELSE IF I_BagInBeam THEN
		Alarm[mySeq].Name = almSwitchFault
	ENDIF
ENDIF

;Step 3 bag settles in weigh beam
TON_10ms(I_BagInBeam,SettleTime,BagSettled,BagSettledET)
IF (STEP = 3) THEN
	IF BagSettled AND (Bag[myBag].Cat > 0) AND (ReportLoading[myLP].Cat = 0) THEN
		Bag[myBag].Wgt = Wgt/10

		ReportLoading[myLP].Prg = Bag[myBag].Prg 			;Program
		ReportLoading[myLP].Cat = Bag[myBag].Cat			;Category
		ReportLoading[myLP].Cus = Bag[myBag].Cus			;Customer
		ReportLoading[myLP].Wgt = Bag[myBag].Wgt			;Weight
		ReportLoading[myLP].Cnt = 0							;Count
		ReportLoading[myLP].Stn = myLP         			;Station
		ReportLoading[myLP].Mcn = 0						;Machine
		ReportLoading[myLP].Bid = Bag[myBag].Bid			;Batch ID
		D[900 + mySeq] = 4
	ELSE IF NOT BagSettled THEN
		Alarm[mySeq].Name = almBagNotSettled
	ELSE IF (Bag[myBag].Cat = 0) THEN
		Alarm[mySeq].Name = almBagDataError
	ELSE IF (ReportLoading[myLP].Cat > 0) THEN
		Alarm[mySeq].Name = almGeneralSequence
	ENDIF
ENDIF

OkToRelease = (Bag[myBag].Cat > 0) AND Line[myRelLine].Clear  AND NOT Line[myRelLine].TripFault
;Step 4 Check for line space
IF (STEP = 4) THEN
	IF OkToRelease THEN
		D[900 + mySeq]  = 5
	ELSE IF (Bag[myBag].Cat = 0) THEN
		Alarm[mySeq].Name = almBagDataError
	ELSE IF Line[myRelLine].TripFault THEN
		Alarm[mySeq].Name = almSwitchFault
	ENDIF
ENDIF

;Step 5 Release Bag
IF (STEP = 5) THEN
	O_OpenSep = OkToRelease
	IF Line[myRelLine].Trip THEN
		Bag[myOutBag] = Bag[myBag]
		Bag[myBag] = Bag[0]
		D[900 + mySeq] = 1
	ENDIF
	IF (Bag[myBag].Cat = 0) THEN
		Alarm[mySeq].Name = almBagDataError
	ELSE IF Line[myRelLine].TripFault THEN
		Alarm[mySeq].Name = almSwitchFault
	ENDIF
ENDIF

;-----------------------------------
;PLC Outputs - adjust to suit system
;-----------------------------------

Y[myIO].Y05 = O_OpenSep

;Alarms
TimerAlarm.IN 		= NOT PLS AND (Alarm[mySeq].Name > 0)
TimerAlarm.PT 		= Alarm[mySeq].Time
TimerAlarm FUB TON_10ms()
Alarm[mySeq].On 	= TimerAlarm.Q
Alarm[mySeq].ET 	= TimerAlarm.ET
Alarm[mySeq].Zone 	= myZone
END_PROGRAM
```

### Program Logical/Reference/8_pwb3 (IEC) - *PWB3 Weigh beam 3

#### pwb.ab
```automation-basic
;--------------------------------------------
;Sequence 0 - XXX0  D[900 + mySeq]
;--------------------------------------------

PROGRAM _INIT
(* init program *)
END_PROGRAM

PROGRAM _CYCLIC

;Inputs
mySeq				= 8	;Sequence number
myIO				= 339
myBag				= 786
myRelLine			= 60
myLP				= 3
myDisplayBag		= myBag
myZone				= 3

myOutBag			= Line[myRelLine].LastBag

SettleTime			= 300

I_BagInBeam			= X[myIO].X02

O_OpenSep			= FALSE

EnableRel.LP[myLP]	= FALSE

Alarm[mySeq].Name 	= 0
Alarm[mySeq].Bag	= myBag
Alarm[mySeq].Beacon	= TRUE
Alarm[mySeq].Extra	= 0
Alarm[mySeq].Time	= 3000

RawWgt = DINT(AI1223Raw[myLP])
RawWgt = (RawWgt * 2000)
IF (RawWgt > 0) THEN
	Wgt = INT(RawWgt / 32767)
ELSE
	Wgt = 0
ENDIF
IF (myBag <> myDisplayBag) THEN
	Bag[myDisplayBag].Cat = 1
	Bag[myDisplayBag].Wgt = Wgt
ENDIF

;Setup Sequence
STEP = D[900 + mySeq]
;Setup Pulse contact
PLS = (STEP <> LASTSTEP)
LASTSTEP = STEP

;Sequence
IF (STEP = 0) THEN
	;Disabled
ENDIF
WeighBeamClear = (Bag[myBag].Cat = 0) AND NOT I_BagInBeam

;Step 1 Check Weigh beam is clear
IF (STEP = 1) THEN
	IF (WeighBeamClear AND NOT Std.HaltSysZone[myZone])  THEN
		D[900 + mySeq]  = 2
	ELSE IF (Bag[myBag].Cat > 0) THEN
		Alarm[mySeq].Name = almBagDataError
	ELSE IF I_BagInBeam THEN
		Alarm[mySeq].Name = almSwitchFault
	ENDIF
ENDIF

;Step 2 Enable Release from Loading point
IF (STEP = 2) THEN
	EnableRel.LP[myLP] = WeighBeamClear
	IF I_BagInBeam AND (Bag[myBag].Cat > 0) THEN
		D[900 + mySeq] = 3
	ELSE IF (Bag[myBag].Cat > 0) THEN
		Alarm[mySeq].Name = almBagDataError
	ELSE IF I_BagInBeam THEN
		Alarm[mySeq].Name = almSwitchFault
	ENDIF
ENDIF

;Step 3 bag settles in weigh beam
TON_10ms(I_BagInBeam,SettleTime,BagSettled,BagSettledET)
IF (STEP = 3) THEN
	IF BagSettled AND (Bag[myBag].Cat > 0) AND (ReportLoading[myLP].Cat = 0) THEN
		Bag[myBag].Wgt = Wgt/10

		ReportLoading[myLP].Prg = Bag[myBag].Prg 			;Program
		ReportLoading[myLP].Cat = Bag[myBag].Cat			;Category
		ReportLoading[myLP].Cus = Bag[myBag].Cus			;Customer
		ReportLoading[myLP].Wgt = Bag[myBag].Wgt			;Weight
		ReportLoading[myLP].Cnt = 0							;Count
		ReportLoading[myLP].Stn = myLP         			;Station
		ReportLoading[myLP].Mcn = 0						;Machine
		ReportLoading[myLP].Bid = Bag[myBag].Bid			;Batch ID
		D[900 + mySeq] = 4
	ELSE IF NOT BagSettled THEN
		Alarm[mySeq].Name = almBagNotSettled
	ELSE IF (Bag[myBag].Cat = 0) THEN
		Alarm[mySeq].Name = almBagDataError
	ELSE IF (ReportLoading[myLP].Cat > 0) THEN
		Alarm[mySeq].Name = almGeneralSequence
	ENDIF
ENDIF

OkToRelease = (Bag[myBag].Cat > 0) AND Line[myRelLine].Clear  AND NOT Line[myRelLine].TripFault
;Step 4 Check for line space
IF (STEP = 4) THEN
	IF OkToRelease THEN
		D[900 + mySeq]  = 5
	ELSE IF (Bag[myBag].Cat = 0) THEN
		Alarm[mySeq].Name = almBagDataError
	ELSE IF Line[myRelLine].TripFault THEN
		Alarm[mySeq].Name = almSwitchFault
	ENDIF
ENDIF

;Step 5 Release Bag
IF (STEP = 5) THEN
	O_OpenSep = OkToRelease
	IF Line[myRelLine].Trip THEN
		Bag[myOutBag] = Bag[myBag]
		Bag[myBag] = Bag[0]
		D[900 + mySeq] = 1
	ENDIF
	IF (Bag[myBag].Cat = 0) THEN
		Alarm[mySeq].Name = almBagDataError
	ELSE IF Line[myRelLine].TripFault THEN
		Alarm[mySeq].Name = almSwitchFault
	ENDIF
ENDIF

;-----------------------------------
;PLC Outputs - adjust to suit system
;-----------------------------------

Y[myIO].Y05 = O_OpenSep

;Alarms
TimerAlarm.IN 		= NOT PLS AND (Alarm[mySeq].Name > 0)
TimerAlarm.PT 		= Alarm[mySeq].Time
TimerAlarm FUB TON_10ms()
Alarm[mySeq].On 	= TimerAlarm.Q
Alarm[mySeq].ET 	= TimerAlarm.ET
Alarm[mySeq].Zone 	= myZone
END_PROGRAM
```

### Program Logical/Reference/10_pup2 (IEC) - *PUP2 Unloading point

#### pup.var
```iecst
VAR RETAIN
	LASTSTEP : UINT;
	PLS : BOOL;
	STEP : UINT;
END_VAR
VAR
	TimerAlarm : TON_10ms;
	mySeq : UINT;
	myIO : UINT;
	I_ReleasePB : BOOL;
	I_UnloadingPointOn : BOOL;
	I_TrolleyReleased : BOOL;
	myBag : UINT;
	O_Lamp : BOOL;
	O_OpenBuffer : BOOL;
	O_Release : BOOL;
	myPup : UINT;
	SettledBuffer : BOOL;
	SettledBufferET : UDINT;
	PUPValid : BOOL;
	myZone : INT;
END_VAR
```

#### pup.ab
```automation-basic
;--------------------------------------------
;Sequence 0 - XXX0  D[900 + mySeq]
;--------------------------------------------

PROGRAM _INIT
(* init program *)
END_PROGRAM

PROGRAM _CYCLIC

;Inputs
mySeq				= 10	;Sequence number
myIO				= 346
myBag				= 988
myPup				= 2
myZone	= 0

I_UnloadingPointOn	= X[myIO].X03
I_ReleasePB			= X[myIO].X04
I_TrolleyReleased	= X[myIO].X08 ; Also Line full

;O_Lamp				= FALSE
PUP[myPup].WorkingLamp = FALSE
O_OpenBuffer		= FALSE
O_Release			= FALSE
Request.UP[myPup]	= FALSE

Alarm[mySeq].Name 	= 0
Alarm[mySeq].Bag	= myBag
Alarm[mySeq].Beacon	= TRUE
Alarm[mySeq].Extra	= 0
Alarm[mySeq].Time	= 3000

PUP[myPup].Enabled = (D[mySeq] > 0) AND I_UnloadingPointOn

IF PUP[myPup].Enabled THEN
	PUP[myPup].WorkingLamp = TRUE ; Lamp will display the Unloading point is turned on and flash when off but bags still in transit
ELSE IF (UnloadingBuffer[myPup].CountBIT > 0) THEN
	PUP[myPup].WorkingLamp = Std.Clock1s
ENDIF
O_Lamp = PUP[myPup].WorkingLamp

;Setup Sequence
STEP = D[900 + mySeq]
;Setup Pulse contact
PLS = (STEP <> LASTSTEP)
LASTSTEP = STEP

;Sequence
IF (STEP = 0) THEN
	;Disabled
ENDIF

;Step 1 Request a bag from PP
IF (STEP = 1) THEN
	PUPValid = (PUP[myPup].Enabled AND (Bag[myBag].Cat = 0) AND NOT Std.HaltSysZone[myZone])
	Request.UP[myPup] = PUPValid
	IF (Bag[myBag].Cat > 0) AND NOT I_ReleasePB THEN
		D[900 + mySeq] = 2
	ENDIF
ENDIF

;Step 2 wait for pushbutton to request release of trolley
IF (STEP = 2) THEN
	IF I_ReleasePB AND (ReportUnloading[myPup].Cat = 0) THEN
		ReportUnloading[myPup].Prg = Bag[myBag].Prg 		;Program
		ReportUnloading[myPup].Cat = Bag[myBag].Cat		;Category
		ReportUnloading[myPup].Cus = Bag[myBag].Cus		;Customer
		ReportUnloading[myPup].Wgt = Bag[myBag].Wgt		;Weight
		ReportUnloading[myPup].Cnt = 0					;Count
		ReportUnloading[myPup].Stn = 0					;Station
		ReportUnloading[myPup].Mcn = myPup				;Machine
		ReportUnloading[myPup].Mis = Bag[myBag].Mis		;Batch ID

		Bag[myBag].Cat = Std.MaxCats
		Bag[myBag].Prg = Std.MaxProg
		Bag[myBag].Cus = Std.MaxCust
		D[900 + mySeq] = 3
	ELSE IF (ReportUnloading[myPup].Cat > 0) THEN
		Alarm[mySeq].Name = almGeneralSequence
	ENDIF
ENDIF

;STEP 3 Check for space in empty trolley buffer.
IF (STEP = 3) THEN
	IF NOT I_TrolleyReleased AND NOT Std.HaltSysZone[myZone] THEN
		D[900 + mySeq] = 4
	ENDIF
ENDIF

;STEP 4 Release trolley
IF (STEP = 4) THEN
	O_Release = TRUE
	IF 	I_TrolleyReleased THEN
		Bag[myBag] = Bag[0]
		D[900 + mySeq] = 1
	ENDIF
	Alarm[mySeq].Name = almBagNotReleased
ENDIF

;-----------------------------------
;PLC Outputs - adjust to suit system
;-----------------------------------

Y[myIO].Y06 = O_Release
Y[myIO].Y07 = O_Lamp

;Alarms
TimerAlarm.IN 		= NOT PLS AND (Alarm[mySeq].Name > 0)
TimerAlarm.PT 		= Alarm[mySeq].Time
TimerAlarm FUB TON_10ms()
Alarm[mySeq].On 	= TimerAlarm.Q
Alarm[mySeq].ET 	= TimerAlarm.ET
Alarm[mySeq].Zone 	= myZone
END_PROGRAM
```

### Program Logical/Reference/11_pup3 (IEC) - *PUP3 Unloading point

#### pup.ab
```automation-basic
;--------------------------------------------
;Sequence 0 - XXX0  D[900 + mySeq]
;--------------------------------------------

PROGRAM _INIT
(* init program *)
END_PROGRAM

PROGRAM _CYCLIC

;Inputs
mySeq				= 11	;Sequence number
myIO				= 347
myBag				= 989
myPup				= 3
myZone	= 0

I_UnloadingPointOn	= X[myIO].X03
I_ReleasePB			= X[myIO].X04
I_TrolleyReleased	= X[myIO].X08 ; Also Line full

;O_Lamp				= FALSE
PUP[myPup].WorkingLamp = FALSE
O_OpenBuffer		= FALSE
O_Release			= FALSE
Request.UP[myPup]	= FALSE

Alarm[mySeq].Name 	= 0
Alarm[mySeq].Bag	= myBag
Alarm[mySeq].Beacon	= TRUE
Alarm[mySeq].Extra	= 0
Alarm[mySeq].Time	= 3000

PUP[myPup].Enabled = (D[mySeq] > 0) AND I_UnloadingPointOn

IF PUP[myPup].Enabled THEN
	PUP[myPup].WorkingLamp = TRUE ; Lamp will display the Unloading point is turned on and flash when off but bags still in transit
ELSE IF (UnloadingBuffer[myPup].CountBIT > 0) THEN
	PUP[myPup].WorkingLamp = Std.Clock1s
ENDIF
O_Lamp = PUP[myPup].WorkingLamp

;Setup Sequence
STEP = D[900 + mySeq]
;Setup Pulse contact
PLS = (STEP <> LASTSTEP)
LASTSTEP = STEP

;Sequence
IF (STEP = 0) THEN
	;Disabled
ENDIF

;Step 1 Request a bag from PP
IF (STEP = 1) THEN
	PUPValid = (PUP[myPup].Enabled AND (Bag[myBag].Cat = 0) AND NOT Std.HaltSysZone[myZone])
	Request.UP[myPup] = PUPValid
	IF (Bag[myBag].Cat > 0) AND NOT I_ReleasePB THEN
		D[900 + mySeq] = 2
	ENDIF
ENDIF

;Step 2 wait for pushbutton to request release of trolley
IF (STEP = 2) THEN
	IF I_ReleasePB AND (ReportUnloading[myPup].Cat = 0) THEN
		ReportUnloading[myPup].Prg = Bag[myBag].Prg 		;Program
		ReportUnloading[myPup].Cat = Bag[myBag].Cat		;Category
		ReportUnloading[myPup].Cus = Bag[myBag].Cus		;Customer
		ReportUnloading[myPup].Wgt = Bag[myBag].Wgt		;Weight
		ReportUnloading[myPup].Cnt = 0					;Count
		ReportUnloading[myPup].Stn = 0					;Station
		ReportUnloading[myPup].Mcn = myPup				;Machine
		ReportUnloading[myPup].Mis = Bag[myBag].Mis		;Batch ID

		Bag[myBag].Cat = Std.MaxCats
		Bag[myBag].Prg = Std.MaxProg
		Bag[myBag].Cus = Std.MaxCust
		D[900 + mySeq] = 3
	ELSE IF (ReportUnloading[myPup].Cat > 0) THEN
		Alarm[mySeq].Name = almGeneralSequence
	ENDIF
ENDIF

;STEP 3 Check for space in empty trolley buffer.
IF (STEP = 3) THEN
	IF NOT I_TrolleyReleased AND NOT Std.HaltSysZone[myZone] THEN
		D[900 + mySeq] = 4
	ENDIF
ENDIF

;STEP 4 Release trolley
IF (STEP = 4) THEN
	O_Release = TRUE
	IF 	I_TrolleyReleased THEN
		Bag[myBag] = Bag[0]
		D[900 + mySeq] = 1
	ENDIF
	Alarm[mySeq].Name = almBagNotReleased
ENDIF

;-----------------------------------
;PLC Outputs - adjust to suit system
;-----------------------------------

Y[myIO].Y06 = O_Release
Y[myIO].Y07 = O_Lamp

;Alarms
TimerAlarm.IN 		= NOT PLS AND (Alarm[mySeq].Name > 0)
TimerAlarm.PT 		= Alarm[mySeq].Time
TimerAlarm FUB TON_10ms()
Alarm[mySeq].On 	= TimerAlarm.Q
Alarm[mySeq].ET 	= TimerAlarm.ET
Alarm[mySeq].Zone 	= myZone
END_PROGRAM
```

### Program Logical/Reference/14_pup6 (IEC) - *PUP6 Unloading point

#### pup.ab
```automation-basic
;--------------------------------------------
;Sequence 0 - XXX0  D[900 + mySeq]
;--------------------------------------------

PROGRAM _INIT
(* init program *)
END_PROGRAM

PROGRAM _CYCLIC

;Inputs
mySeq				= 14	;Sequence number
myIO				= 350
myBag				= 999
myPup				= 6
myZone	= 0

I_UnloadingPointOn	= X[myIO].X03
I_ReleasePB			= X[myIO].X04
I_TrolleyReleased	= X[myIO].X08 ; Also Line full

;O_Lamp				= FALSE
PUP[myPup].WorkingLamp = FALSE
O_OpenBuffer		= FALSE
O_Release			= FALSE
Request.UP[myPup]	= FALSE

Alarm[mySeq].Name 	= 0
Alarm[mySeq].Bag	= myBag
Alarm[mySeq].Beacon	= TRUE
Alarm[mySeq].Extra	= 0
Alarm[mySeq].Time	= 3000

PUP[myPup].Enabled = (D[mySeq] > 0) AND I_UnloadingPointOn

IF PUP[myPup].Enabled THEN
	PUP[myPup].WorkingLamp = TRUE ; Lamp will display the Unloading point is turned on and flash when off but bags still in transit
ELSE IF (UnloadingBuffer[myPup].CountBIT > 0) THEN
	PUP[myPup].WorkingLamp = Std.Clock1s
ENDIF
O_Lamp = PUP[myPup].WorkingLamp

;Setup Sequence
STEP = D[900 + mySeq]
;Setup Pulse contact
PLS = (STEP <> LASTSTEP)
LASTSTEP = STEP

;Sequence
IF (STEP = 0) THEN
	;Disabled
ENDIF

;Step 1 Request a bag from PP
IF (STEP = 1) THEN
	PUPValid = (PUP[myPup].Enabled AND (Bag[myBag].Cat = 0) AND NOT Std.HaltSysZone[myZone])
	Request.UP[myPup] = PUPValid
	IF (Bag[myBag].Cat > 0) AND NOT I_ReleasePB THEN
		D[900 + mySeq] = 2
	ENDIF
ENDIF

;Step 2 wait for pushbutton to request release of trolley
IF (STEP = 2) THEN
	IF I_ReleasePB AND (ReportUnloading[myPup].Cat = 0) THEN
		ReportUnloading[myPup].Prg = Bag[myBag].Prg 		;Program
		ReportUnloading[myPup].Cat = Bag[myBag].Cat		;Category
		ReportUnloading[myPup].Cus = Bag[myBag].Cus		;Customer
		ReportUnloading[myPup].Wgt = Bag[myBag].Wgt		;Weight
		ReportUnloading[myPup].Cnt = 0					;Count
		ReportUnloading[myPup].Stn = 0					;Station
		ReportUnloading[myPup].Mcn = myPup				;Machine
		ReportUnloading[myPup].Mis = Bag[myBag].Mis		;Batch ID

		Bag[myBag].Cat = Std.MaxCats
		Bag[myBag].Prg = Std.MaxProg
		Bag[myBag].Cus = Std.MaxCust
		D[900 + mySeq] = 3
	ELSE IF (ReportUnloading[myPup].Cat > 0) THEN
		Alarm[mySeq].Name = almGeneralSequence
	ENDIF
ENDIF

;STEP 3 Check for space in empty trolley buffer.
IF (STEP = 3) THEN
	IF NOT I_TrolleyReleased AND NOT Std.HaltSysZone[myZone] THEN
		D[900 + mySeq] = 4
	ENDIF
ENDIF

;STEP 4 Release trolley
IF (STEP = 4) THEN
	O_Release = TRUE
	IF 	I_TrolleyReleased THEN
		Bag[myBag] = Bag[0]
		D[900 + mySeq] = 1
	ENDIF
	Alarm[mySeq].Name = almBagNotReleased
ENDIF

;-----------------------------------
;PLC Outputs - adjust to suit system
;-----------------------------------

Y[myIO].Y06 = O_Release
Y[myIO].Y07 = O_Lamp

;Alarms
TimerAlarm.IN 		= NOT PLS AND (Alarm[mySeq].Name > 0)
TimerAlarm.PT 		= Alarm[mySeq].Time
TimerAlarm FUB TON_10ms()
Alarm[mySeq].On 	= TimerAlarm.Q
Alarm[mySeq].ET 	= TimerAlarm.ET
Alarm[mySeq].Zone 	= myZone
END_PROGRAM
```

- Program Logical/Reference/15_pbr1 (IEC, version 1.00.0) - *PBR1 Bag Remover (no source held here)

### Program Logical/Reference/16_pbr2 (IEC) - *PBR2 Bag Remover

#### pbr.ab
```automation-basic
PROGRAM _INIT
	(* init program *)
END_PROGRAM

PROGRAM _CYCLIC
	(* cyclic program *)

;Sequence 1- Primary Bag remover 1 D[900 + mySeq]

;-----------------------------------------
;Revision 1.00 12/11/2002 D.J. First Issue
;-----------------------------------------
mySeq   = 16
myIO	= 252
myPbr	= 2
myZone	= 0

I_BagAtSeparator	= X[myIO].X01
I_BagAtRemover		= X[myIO].X02
I_BagReleased		= X[myIO].X03

O_OpenSeparator		= FALSE
O_Locate			= FALSE
O_OpenStop			= FALSE

;Setup Sequence
;-----------------------
STEP = D[900 + mySeq]
;Setup Pulse contact
PLS = (STEP <> LASTSTEP)
LASTSTEP = STEP

;Alarm
Alarm[mySeq].Name 	= 0
Alarm[mySeq].Bag	= 0
Alarm[mySeq].Beacon	= TRUE
Alarm[mySeq].Extra	= 0
Alarm[mySeq].Time	= 3000

;Sequence
IF (STEP = 0) THEN
	;Disabled
ENDIF

;Wait for bag at separator
IF (STEP = 1) THEN
	O_OpenSeparator = TRUE
	IF I_BagAtRemover THEN
		D[900 + mySeq] = 3
	ELSE IF I_BagAtSeparator THEN
		D[900 + mySeq] = 2
	ENDIF
ENDIF

;Open separator
;Was 3 seconds
TON_10ms((STEP = 2),50,SeparatorOpened,SeparatorOpenedET)
IF (STEP = 2) THEN
	;O_OpenSeparator = TRUE
	IF SeparatorOpened THEN
		D[900 + mySeq] = 3
	ENDIF
ENDIF

;Wait for bag at remover
;Was 3.5 Seconds
TON_10ms(I_BagAtRemover,200,SettledAtRemover,SettledAtRemoverET)
TON_10ms((STEP = 3),2000,Step3TimedOut,Step3TimedOutET)
IF (STEP = 3) THEN
	;O_OpenSeparator = TRUE
	IF SettledAtRemover THEN;AND NOT I_BagReleased) THEN
		D[900 + mySeq] = 4
	ELSE IF Step3TimedOut THEN; AND NOT I_BagReleased) THEN
		D[900 + mySeq] = 1
	ENDIF
ENDIF

;Allow bag to settle
;Was 4 seconds
TON_10ms((STEP = 4),200,Settled,SettledET)
IF (STEP = 4) THEN
	IF (CAN[1].OkToRelease[myPbr] AND Settled AND NOT I_BagReleased) THEN ;(Settled OR I_BagReleased)) THEN
		D[900 + mySeq] = 5
	ENDIF
ENDIF

;Locate hook
;Was 5 seconds
TON_10ms((STEP = 5),300,Located,LocatedET)
IF (STEP = 5) THEN
	O_Locate = TRUE
	IF Located OR I_BagReleased THEN
		D[900 + mySeq] = 6
	ENDIF
ENDIF

;Strip bag
TON_10ms((STEP = 6),1000,Step6TimedOut,Step6TimedOutET)
TON_10ms((STEP = 6),200,RemoveLocate,RemoveLocateET)
IF (STEP = 6) THEN
	O_Locate 	= NOT RemoveLocate
	O_OpenStop 	= TRUE
	IF I_BagReleased THEN
		D[900 + mySeq] = 1
	ELSE IF Step6TimedOut THEN
		D[900 + mySeq] = 4
	ENDIF
ENDIF

;Alarms
TimerAlarm.IN 		= NOT PLS AND (Alarm[mySeq].Name > 0)
TimerAlarm.PT 		= Alarm[mySeq].Time
TimerAlarm FUB TON_10ms()
Alarm[mySeq].On 	= TimerAlarm.Q
Alarm[mySeq].ET 	= TimerAlarm.ET
Alarm[mySeq].Zone 	= myZone

Y[myIO].Y04 = O_OpenSeparator
Y[myIO].Y06 = O_Locate
Y[myIO].Y05 = O_OpenStop
END_PROGRAM
```

### Program Logical/Reference/17_pp3 (IEC) - *PP3 Full bags to PICD 4&5

#### pp.var
```iecst
VAR
	BagValid : BOOL;
	DestValid : BOOL;
	I_BagAtSep : BOOL;
	I_BagReleased : BOOL;
END_VAR
VAR RETAIN
	LASTSTEP : UINT;
END_VAR
VAR
	myBag : UINT;
	myDest : USINT;
	myIC : USINT;
	myIO : UINT;
	mySeq : UINT;
	O_OpenSep : BOOL;
	O_Select : ARRAY[0..9] OF BOOL;
END_VAR
VAR RETAIN
	PLS : BOOL;
END_VAR
VAR
	PointsReset : BOOL;
	PointsResetET : UDINT;
END_VAR
VAR RETAIN
	myPrevIC : USINT;
END_VAR
VAR
	ResetPoints : BOOL;
	SettledAtSep : BOOL;
	SettledAtSepET : UDINT;
END_VAR
VAR RETAIN
	STEP : UINT;
END_VAR
VAR
	TimerAlarm : TON_10ms;
	BagReleased : BOOL;
	myZone : INT;
	myICBufferBag : ARRAY[0..5] OF UINT;
	I_InclineBufferClear : ARRAY[0..5] OF BOOL;
	ReleaseValid : BOOL;
	InclineClear : BOOL;
	I_BagInSep : BOOL;
	BagInSep : BOOL;
	SettledInSep : BOOL;
	SettledInSepET : UDINT;
	I_BagArriveIC : ARRAY[0..5] OF BOOL;
END_VAR
```

### Program Logical/Reference/19_pp5 (IEC) - *PP5 Full bags to PUP 2&3

#### pp.ab
```automation-basic
;--------------------------------------------
;Sequence 0 - XXX0  D[900 + mySeq]
;--------------------------------------------

PROGRAM _INIT
(* init program *)
END_PROGRAM

PROGRAM _CYCLIC

;Inputs
mySeq				= 19	;Sequence number
myIO				= 105
myBag				= 958

myZone	= 0

myOutBag[1]			= 988
myOutBag[2]			= 989
myRelDest[1]		= 22	;Destination in Bag for PUP 2
myRelDest[2]		= 23

myPUP[1]			= (myRelDest[1] - 20)
myPUP[2]			= (myRelDest[2] - 20)

I_BagAtSep			= X[myIO].X01
I_BagInSep			= X[myIO].X03
I_BagArrive[1]		= X[myIO].X02
I_BagArrive[2]		= X[myIO].X04

AutoDestChange 		= (D[mySeq] > 0)

O_OpenSep			= FALSE
O_Select[1]			= FALSE
O_Select[2]			= FALSE

Alarm[mySeq].Name 	= 0
Alarm[mySeq].Bag	= myBag
Alarm[mySeq].Beacon	= TRUE
Alarm[mySeq].Extra	= 0
Alarm[mySeq].Time	= 3000

;Setup Sequence
STEP = D[900 + mySeq]
;Setup Pulse contact
PLS = (STEP <> LASTSTEP)
LASTSTEP = STEP

TON_10ms(I_BagInSep,75,SettledInSep,SettledInSepET)
IF (STEP < 2) THEN
	BagInSep = FALSE
ELSE IF SettledInSep THEN
	BagInSep = TRUE
ENDIF

;Sequence
IF (STEP = 0) THEN
	;Disabled
ENDIF

;step 1 Check destination of bag in buffer
myDest = Bag[myBag].Dst
BagValid = (Bag[myBag].Cat > 0)
PUPClear[1] = (Bag[myOutBag[1]].Cat = 0)
PUPClear[2] = (Bag[myOutBag[2]].Cat = 0)

TON_10ms(I_BagAtSep,75,SettledAtSep,SettledAtSepET)
TON_10ms(ResetPoints,100,PointsReset,PointsResetET)
IF (STEP = 1) THEN
	IF (myDest = myRelDest[1]) THEN
		mySelLine = 1
	ELSE IF	(myDest = myRelDest[2]) THEN
		mySelLine = 2
	ELSE
		mySelLine = 0
	ENDIF
	DestValid = (mySelLine > 0)
	IF BagValid AND DestValid AND SettledAtSep AND NOT I_BagInSep THEN
		IF (mySelLine = myPrevSelLine) AND DestValid THEN
			IF (myDest = myRelDest[1]) AND PUPClear[1] THEN
				D[900 + mySeq]  = 2
			ELSE IF (myDest = myRelDest[2]) THEN
				D[900 + mySeq]  = 4
			ENDIF
		ELSE
			ResetPoints = TRUE
			IF (myDest= myRelDest[1]) THEN
				O_Select[1] = TRUE
				IF PointsReset THEN
					D[900 + mySeq]  = 2
				ENDIF
			ELSE IF (myDest= myRelDest[2]) THEN
				O_Select[2] = TRUE
				IF PointsReset THEN
					D[900 + mySeq]  = 4
				ENDIF
			ENDIF
		ENDIF
	ENDIF
	IF NOT BagValid	AND SettledAtSep THEN
		Alarm[mySeq].Name = almBagDataError
	ELSE IF BagValid AND NOT SettledAtSep THEN
		Alarm[mySeq].Name = almSwitchFault
	ELSE IF NOT DestValid AND SettledAtSep THEN
		Alarm[mySeq].Time = 0
		Alarm[mySeq].Name = almDestinationNotValid
	ENDIF
ELSE
	ResetPoints = FALSE
ENDIF

;Step 2 Wait for enable from PUP
IF (STEP = 2) THEN
	mySelLine = 1
	myPrevSelLine = mySelLine
	IF AutoDestChange AND Request.UP[myPUP[2]] AND PUPClear[2] AND NOT PUP[myPUP[mySelLine]].Enabled  THEN ; If the selected PUP is turned Off - Automatically route the bags to the other Discharger...
		Bag[myBag].Dst	= myRelDest[2]
		GOTO ExitSeq
	ENDIF
	DestValid = (myDest = myRelDest[mySelLine])
	O_Select[mySelLine] = DestValid AND PUPClear[mySelLine]
	IF NOT DestValid THEN ; Destination has been changed..
		D[900 + mySeq] = 1
	ELSE IF (Request.UP[myPUP[mySelLine]] AND PUPClear[mySelLine] AND DestValid AND BagValid AND SettledAtSep AND NOT I_BagArrive[mySelLine] AND NOT Std.HaltSysZone[myZone]) THEN
		D[900 + mySeq] = 3
	ENDIF
	IF Request.IC[mySelLine] AND NOT PUPClear[mySelLine] THEN
		Alarm[mySeq].Bag = myOutBag[mySelLine]
		Alarm[mySeq].Name = almBagDataError
	ELSE IF I_BagArrive[mySelLine] THEN
		Alarm[mySeq].Name = almSwitchFault
	ELSE IF NOT BagValid	AND SettledAtSep THEN
		Alarm[mySeq].Name = almBagDataError
	ELSE IF BagValid AND NOT SettledAtSep THEN
		Alarm[mySeq].Name = almSwitchFault
	ELSE IF NOT Std.HaltSysZone[myZone] THEN
	;	Alarm[mySeq].Name = almBagNotReleased
	ENDIF
ENDIF

;Step 3 Release bag to PUP
IF (STEP = 3) THEN
	mySelLine = 1
	myPrevSelLine = mySelLine
	DestValid = (myDest = myRelDest[mySelLine])
	O_Select[mySelLine] = DestValid
	IF (Request.UP[myPUP[mySelLine]] AND DestValid AND BagValid AND PUPClear[mySelLine] AND NOT I_BagArrive[mySelLine]) THEN
		ReleaseValid = TRUE
	ENDIF
	O_OpenSep = ReleaseValid AND NOT BagInSep
	IF I_BagArrive[mySelLine] AND PUPClear[mySelLine] AND BagValid THEN
		Bag[myOutBag[mySelLine]] = Bag[myBag]
		Bag[myBag] = Bag[0]
		D[900 + mySeq] = 1
	ENDIF
	IF NOT PUPClear[mySelLine] THEN
		Alarm[mySeq].Bag = myOutBag[mySelLine]
		Alarm[mySeq].Name = almBagDataError
	ELSE IF NOT BagValid AND SettledAtSep THEN
		Alarm[mySeq].Name = almBagDataError
	ELSE IF BagValid AND NOT SettledAtSep THEN
		Alarm[mySeq].Name = almSwitchFault
	ELSE IF NOT DestValid AND SettledAtSep THEN
		Alarm[mySeq].Name = almDestinationNotValid
	ENDIF
ELSE
	ReleaseValid = FALSE
ENDIF

;Step 4 Wait for enable from PUP
IF (STEP = 4) THEN
	mySelLine = 2
	myPrevSelLine = mySelLine
	IF AutoDestChange AND Request.UP[myPUP[1]] AND PUPClear[1] AND NOT PUP[myPUP[mySelLine]].Enabled THEN ; If the selected PUP is turned Off - Automatically route the bags to the other Discharger...
		Bag[myBag].Dst	= myRelDest[1]
		GOTO ExitSeq
	ENDIF
	DestValid = (myDest = myRelDest[mySelLine])
	O_Select[mySelLine] = DestValid AND PUPClear[mySelLine]
	IF NOT DestValid THEN ; Destination has been changed..
		D[900 + mySeq] = 1
	ELSE IF (Request.UP[myPUP[mySelLine]] AND PUPClear[mySelLine] AND DestValid AND BagValid AND SettledAtSep AND NOT I_BagArrive[mySelLine] AND NOT Std.HaltSysZone[myZone]) THEN
		D[900 + mySeq] = 5
	ENDIF
	IF Request.IC[mySelLine] AND NOT PUPClear[mySelLine] THEN
		Alarm[mySeq].Bag = myOutBag[mySelLine]
		Alarm[mySeq].Name = almBagDataError
	ELSE IF I_BagArrive[mySelLine] THEN
		Alarm[mySeq].Name = almSwitchFault
	ELSE IF NOT BagValid	AND SettledAtSep THEN
		Alarm[mySeq].Name = almBagDataError
	ELSE IF BagValid AND NOT SettledAtSep THEN
		Alarm[mySeq].Name = almSwitchFault
	ELSE IF NOT Std.HaltSysZone[myZone] THEN
	;	Alarm[mySeq].Name = almBagNotReleased
	ENDIF
ENDIF

;Step 5 Release bag to PUP
IF (STEP = 5) THEN
	mySelLine = 2
	myPrevSelLine = mySelLine
	DestValid = (myDest = myRelDest[mySelLine])
	O_Select[mySelLine] = DestValid
	O_OpenSep = (Request.UP[myPUP[mySelLine]] AND DestValid AND BagValid AND PUPClear[mySelLine] AND NOT BagInSep AND NOT I_BagArrive[mySelLine])
	IF I_BagArrive[mySelLine] AND PUPClear[mySelLine] AND BagValid THEN
		Bag[myOutBag[mySelLine]] = Bag[myBag]
		Bag[myBag] = Bag[0]
		D[900 + mySeq] = 1
	ENDIF
	IF NOT PUPClear[mySelLine] THEN
		Alarm[mySeq].Bag = myOutBag[mySelLine]
		Alarm[mySeq].Name = almBagDataError
	ELSE IF NOT BagValid AND SettledAtSep THEN
		Alarm[mySeq].Name = almBagDataError
	ELSE IF BagValid AND NOT SettledAtSep THEN
		Alarm[mySeq].Name = almSwitchFault
	ELSE IF NOT DestValid AND SettledAtSep THEN
		Alarm[mySeq].Name = almDestinationNotValid
	ENDIF
ENDIF
;-----------------------------------
;PLC Outputs - adjust to suit system
;-----------------------------------

ExitSeq:

Y[myIO].Y05 = O_OpenSep
Y[myIO].Y07 = O_Select[2]
Y[myIO].Y08 = O_Select[1]

;Alarms
TimerAlarm.IN 		= NOT PLS AND (Alarm[mySeq].Name > 0)
TimerAlarm.PT 		= Alarm[mySeq].Time
TimerAlarm FUB TON_10ms()
Alarm[mySeq].On 	= TimerAlarm.Q
Alarm[mySeq].ET 	= TimerAlarm.ET
Alarm[mySeq].Zone 	= myZone
END_PROGRAM
```

### Program Logical/Reference/20_pp6 (IEC) - *PP6 Empty trolleys feeding PICU7

#### pp.var
```iecst
VAR RETAIN
	LASTSTEP : UINT;
	PLS : BOOL;
	STEP : UINT;
END_VAR
VAR
	TimerAlarm : TON_10ms;
	mySeq : UINT;
	myIO : UINT;
	I_BagAtSep : ARRAY[0..2] OF BOOL;
	I_LineFull : BOOL;
	O_OpenSep : ARRAY[0..2] OF BOOL;
	O_Select : ARRAY[0..2] OF BOOL;
	SettledAtSep : ARRAY[0..2] OF BOOL;
	SettledAtSepET : ARRAY[0..2] OF UDINT;
	myLine : USINT;
	TrolleyCount : ARRAY[0..2] OF UINT;
	TrolleyBatchSize : UINT;
	n : UINT;
	I_BufferLineFull : ARRAY[0..2] OF BOOL;
	BufferFull : ARRAY[0..2] OF BOOL;
	BufferFullET : ARRAY[0..2] OF UDINT;
	Reset : BOOL;
	ResetPoints : BOOL;
	ResetPointsET : UDINT;
END_VAR
VAR RETAIN
	myPrevLine : UINT;
END_VAR
VAR
	myZone : INT;
	I_BagInSep : ARRAY[0..3] OF BOOL;
	SettledInSep : ARRAY[0..2] OF BOOL;
	SettledInSepET : ARRAY[0..2] OF UDINT;
	BagInSep : BOOL;
END_VAR
```

### Program Logical/Reference/21_pp7 (IEC) - *PP7 Empty trolleys from PUP 1-3

#### pp.ab
```automation-basic
;--------------------------------------------
;Sequence 0 - XXX0  D[900 + mySeq]
;--------------------------------------------

PROGRAM _INIT
(* init program *)
END_PROGRAM

PROGRAM _CYCLIC

;Inputs
mySeq				= 21	;Sequence number
myIO				= 107
myZone	= 0

TrolleyBatchSize 	= 4

I_BagAtSep[1]			= X[myIO].X01
I_BagAtSep[2]			= X[myIO].X02
I_BagInSep[1]			= X[347].X01
I_BagInSep[2]			= X[347].X02
I_LineFull				= X[myIO].X03
I_BufferLineFull[1]		= X[347].X08
I_BufferLineFull[2]		= X[177].X05

O_OpenSep[1]			= FALSE
O_OpenSep[2]			= FALSE
O_Select[1]				= FALSE
O_Select[2]				= FALSE

Alarm[mySeq].Name 	= 0
Alarm[mySeq].Bag	= 10000 + mySeq
Alarm[mySeq].Beacon	= TRUE
Alarm[mySeq].Extra	= 0
Alarm[mySeq].Time	= 3000

;Setup Sequence
STEP = D[900 + mySeq]
;Setup Pulse contact
PLS = (STEP <> LASTSTEP)
LASTSTEP = STEP

;Keep trolley counts inrange
LOOP n = 1 TO 2 DO
	IF (TrolleyCount[n] >$FFFE) THEN
		TrolleyCount[n] = $FFFE
	ENDIF
ENDLOOP

;Sequence
IF (STEP = 0) THEN
	;Disabled
ENDIF

;Step 1 Decide where to take trolley from
TON_10ms(I_BagAtSep[1],200,SettledAtSep[1],SettledAtSepET[1])
TON_10ms(I_BagAtSep[2],200,SettledAtSep[2],SettledAtSepET[2])
TON_10ms(I_BufferLineFull[1],400,BufferFull[1],BufferFullET[1])
TON_10ms(I_BufferLineFull[2],400,BufferFull[2],BufferFullET[2])
TON_10ms(Reset,200,ResetPoints,ResetPointsET)
IF (STEP = 1) THEN
	;Force line choice if line is full
	IF NOT Reset THEN
		IF BufferFull[1] AND NOT BufferFull[2] THEN
			myLine = 1
		ELSE IF BufferFull[2] AND NOT BufferFull[1] THEN
			myLine = 2
		ENDIF
	ENDIF
	IF (myLine = 0) OR (myLine > 2) THEN
		myLine = 1
	ENDIF

	IF (SettledAtSep[myLine] AND (TrolleyCount[myLine] < TrolleyBatchSize) AND NOT I_LineFull AND NOT Reset AND NOT Std.HaltSysZone[myZone]) THEN
		IF (myLine = myPrevLine) THEN
			D[900 +  mySeq] = (myLine + 1)
		ELSE
			Reset = TRUE
		ENDIF
	ELSE IF Reset THEN
		O_Select[myLine] = TRUE
		IF ResetPoints THEN
			myPrevLine = myLine
			D[900 +  mySeq] = (myLine + 1)
		ENDIF
	ELSE IF (TrolleyCount[myLine] >= TrolleyBatchSize) OR NOT I_BagAtSep[myLine] THEN
		TrolleyCount[myLine] = 0
		INC myLine
	ENDIF
ELSE
	Reset = FALSE
ENDIF

;Step 2 Select Line 1
TON_10ms(I_BagInSep[1],150,SettledInSep[1],SettledInSepET[1])
IF (STEP = 2) THEN
	myLine = 1
	IF SettledInSep[myLine] THEN
		BagInSep[myLine] = TRUE
	ENDIF
	O_Select[myLine] = TRUE
	O_OpenSep[myLine] = NOT BagInSep[myLine]
	IF I_LineFull THEN
		INC TrolleyCount[myLine]
		D[900 + mySeq] = 1
	ENDIF
	Alarm[mySeq].Name = almBagNotReleased
ELSE
	BagInSep[1] = FALSE
ENDIF

;Step 3 Select Line 2
TON_10ms(I_BagInSep[2],150,SettledInSep[2],SettledInSepET[2])
IF (STEP = 3) THEN
	myLine = 2
	IF SettledInSep[myLine] THEN
		BagInSep[myLine] = TRUE
	ENDIF
	O_Select[myLine] = TRUE
	O_OpenSep[myLine] = NOT BagInSep[myLine]
	IF I_LineFull THEN
		INC TrolleyCount[myLine]
		D[900 + mySeq] = 1
	ENDIF
	Alarm[mySeq].Name = almBagNotReleased
ELSE
	BagInSep[2] = FALSE
ENDIF

;-----------------------------------
;PLC Outputs - adjust to suit system
;-----------------------------------

Y[myIO].Y05 = O_OpenSep[1]
Y[myIO].Y06 = O_OpenSep[2]
Y[myIO].Y07 = O_Select[1]
Y[myIO].Y08 = O_Select[2]

;Alarms
TimerAlarm.IN 		= NOT PLS AND (Alarm[mySeq].Name > 0)
TimerAlarm.PT 		= Alarm[mySeq].Time
TimerAlarm FUB TON_10ms()
Alarm[mySeq].On 	= TimerAlarm.Q
Alarm[mySeq].ET 	= TimerAlarm.ET
Alarm[mySeq].Zone 	= myZone
END_PROGRAM

END_PROGRAM
```

### Program Logical/Reference/22_pp8 (IEC) - *PP8 Full bag from PID5

#### pp.var
```iecst
VAR
	BagInSep : BOOL;
	BagValid : BOOL;
	DestValid : BOOL;
	I_BagAtSep : BOOL;
	I_BagInSep : BOOL;
END_VAR
VAR RETAIN
	LASTSTEP : UINT;
END_VAR
VAR
	LineValid : ARRAY[0..2] OF BOOL;
	myBag : UINT;
	myDest : USINT;
	myIO : UINT;
	myIO2 : UINT;
	myPrevSelLine : USINT;
	myRelLastBag : ARRAY[0..2] OF UINT;
	myRelLine : ARRAY[0..2] OF UINT;
	mySelLine : USINT;
	mySeq : UINT;
	myZone : INT;
	O_OpenSep : BOOL;
	O_Select : ARRAY[0..2] OF BOOL;
END_VAR
VAR RETAIN
	PLS : BOOL;
END_VAR
VAR
	PointsReset : BOOL;
	PointsResetET : UDINT;
	ResetPoints : BOOL;
	SettledAtSep : BOOL;
	SettledAtSepET : UDINT;
	SettledInSep : BOOL;
	SettledInSepET : UDINT;
END_VAR
VAR RETAIN
	STEP : UINT;
END_VAR
VAR
	TimerAlarm : TON_10ms;
END_VAR
```

### Program Logical/Reference/23_pp9 (IEC) - *PP9 Full bags to PUP 5&6

#### pp.ab
```automation-basic
;--------------------------------------------
;Sequence 0 - XXX0  D[900 + mySeq]
;--------------------------------------------

PROGRAM _INIT
(* init program *)
END_PROGRAM

PROGRAM _CYCLIC

;Inputs
mySeq				= 23	;Sequence number
myIO				= 109
myBag				= 955
myZone	= 0

myOutBag[1]			= 998
myOutBag[2]			= 999
myRelDest[1]		= 25	;Destination in Bag for PUP 5
myRelDest[2]		= 26

myPUP[1]			= (myRelDest[1] - 20)
myPUP[2]			= (myRelDest[2] - 20)

I_BagAtSep			= X[myIO].X01
I_BagInSep			= X[myIO].X03
I_BagArrive[1]		= X[myIO].X02
I_BagArrive[2]		= X[myIO].X04

AutoDestChange 		= (D[mySeq] > 0)

O_OpenSep			= FALSE
O_Select[1]			= FALSE
O_Select[2]			= FALSE

Alarm[mySeq].Name 	= 0
Alarm[mySeq].Bag	= myBag
Alarm[mySeq].Beacon	= TRUE
Alarm[mySeq].Extra	= 0
Alarm[mySeq].Time	= 3000

;Setup Sequence
STEP = D[900 + mySeq]
;Setup Pulse contact
PLS = (STEP <> LASTSTEP)
LASTSTEP = STEP

TON_10ms(I_BagInSep,75,SettledInSep,SettledInSepET)
IF (STEP < 2) THEN
	BagInSep = FALSE
ELSE IF SettledInSep THEN
	BagInSep = TRUE
ENDIF

;Sequence
IF (STEP = 0) THEN
	;Disabled
ENDIF

;step 1 Check destination of bag in buffer
myDest = Bag[myBag].Dst
BagValid = (Bag[myBag].Cat > 0)
PUPClear[1] = (Bag[myOutBag[1]].Cat = 0)
PUPClear[2] = (Bag[myOutBag[2]].Cat = 0)

TON_10ms(I_BagAtSep,75,SettledAtSep,SettledAtSepET)
TON_10ms(ResetPoints,100,PointsReset,PointsResetET)
IF (STEP = 1) THEN
	IF (myDest = myRelDest[1]) THEN
		mySelLine = 1
	ELSE IF	(myDest = myRelDest[2]) THEN
		mySelLine = 2
	ELSE
		mySelLine = 0
	ENDIF
	DestValid = (mySelLine > 0)
	IF BagValid AND DestValid AND SettledAtSep AND NOT I_BagInSep THEN
		IF (mySelLine = myPrevSelLine) AND DestValid THEN
			IF (myDest = myRelDest[1]) AND PUPClear[1] THEN
				D[900 + mySeq]  = 2
			ELSE IF (myDest = myRelDest[2]) THEN
				D[900 + mySeq]  = 4
			ENDIF
		ELSE
			ResetPoints = TRUE
			IF (myDest= myRelDest[1]) THEN
				O_Select[1] = TRUE
				IF PointsReset THEN
					D[900 + mySeq]  = 2
				ENDIF
			ELSE IF (myDest= myRelDest[2]) THEN
				O_Select[2] = TRUE
				IF PointsReset THEN
					D[900 + mySeq]  = 4
				ENDIF
			ENDIF
		ENDIF
	ENDIF
	IF NOT BagValid	AND SettledAtSep THEN
		Alarm[mySeq].Name = almBagDataError
	ELSE IF BagValid AND NOT SettledAtSep THEN
		Alarm[mySeq].Name = almSwitchFault
	ELSE IF NOT DestValid AND SettledAtSep THEN
		Alarm[mySeq].Time = 0
		Alarm[mySeq].Name = almDestinationNotValid
	ENDIF
ELSE
	ResetPoints = FALSE
ENDIF

;Step 2 Wait for enable from PUP
IF (STEP = 2) THEN
	mySelLine = 1
	myPrevSelLine = mySelLine
	IF AutoDestChange AND Request.UP[myPUP[2]] AND PUPClear[2] AND NOT PUP[myPUP[mySelLine]].Enabled  THEN ; If the selected PUP is turned Off - Automatically route the bags to the other Discharger...
		Bag[myBag].Dst	= myRelDest[2]
		GOTO ExitSeq
	ENDIF
	DestValid = (myDest = myRelDest[mySelLine])
	O_Select[mySelLine] = DestValid AND PUPClear[mySelLine]
	IF NOT DestValid THEN ; Destination has been changed..
		D[900 + mySeq] = 1
	ELSE IF (Request.UP[myPUP[mySelLine]] AND PUPClear[mySelLine] AND DestValid AND BagValid AND SettledAtSep AND NOT I_BagArrive[mySelLine] AND NOT Std.HaltSysZone[myZone]) THEN
		D[900 + mySeq] = 3
	ENDIF
	IF Request.IC[mySelLine] AND NOT PUPClear[mySelLine] THEN
		Alarm[mySeq].Bag = myOutBag[mySelLine]
		Alarm[mySeq].Name = almBagDataError
	ELSE IF I_BagArrive[mySelLine] THEN
		Alarm[mySeq].Name = almSwitchFault
	ELSE IF NOT BagValid	AND SettledAtSep THEN
		Alarm[mySeq].Name = almBagDataError
	ELSE IF BagValid AND NOT SettledAtSep THEN
		Alarm[mySeq].Name = almSwitchFault
	ELSE IF NOT Std.HaltSysZone[myZone] THEN
		;Alarm[mySeq].Name = almBagNotReleased
	ENDIF
ENDIF

;Step 3 Release bag to PUP
IF (STEP = 3) THEN
	mySelLine = 1
	myPrevSelLine = mySelLine
	DestValid = (myDest = myRelDest[mySelLine])
	O_Select[mySelLine] = DestValid
	IF (Request.UP[myPUP[mySelLine]] AND DestValid AND BagValid AND PUPClear[mySelLine] AND NOT I_BagArrive[mySelLine]) THEN
		ReleaseValid = TRUE
	ENDIF
	O_OpenSep = ReleaseValid AND NOT BagInSep
	IF I_BagArrive[mySelLine] AND PUPClear[mySelLine] AND BagValid THEN
		Bag[myOutBag[mySelLine]] = Bag[myBag]
		Bag[myBag] = Bag[0]
		D[900 + mySeq] = 1
	ENDIF
	IF NOT PUPClear[mySelLine] THEN
		Alarm[mySeq].Bag = myOutBag[mySelLine]
		Alarm[mySeq].Name = almBagDataError
	ELSE IF NOT BagValid AND SettledAtSep THEN
		Alarm[mySeq].Name = almBagDataError
	ELSE IF BagValid AND NOT SettledAtSep THEN
		Alarm[mySeq].Name = almSwitchFault
	ELSE IF NOT DestValid AND SettledAtSep THEN
		Alarm[mySeq].Name = almDestinationNotValid
	ENDIF
ELSE
	ReleaseValid = FALSE
ENDIF

;Step 4 Wait for enable from PUP
IF (STEP = 4) THEN
	mySelLine = 2
	myPrevSelLine = mySelLine
	IF AutoDestChange AND Request.UP[myPUP[1]] AND PUPClear[1] AND NOT PUP[myPUP[mySelLine]].Enabled THEN ; If the selected PUP is turned Off - Automatically route the bags to the other Discharger...
		Bag[myBag].Dst	= myRelDest[1]
		GOTO ExitSeq
	ENDIF
	DestValid = (myDest = myRelDest[mySelLine])
	O_Select[mySelLine] = DestValid AND PUPClear[mySelLine]
	IF NOT DestValid THEN ; Destination has been changed..
		D[900 + mySeq] = 1
	ELSE IF (Request.UP[myPUP[mySelLine]] AND PUPClear[mySelLine] AND DestValid AND BagValid AND SettledAtSep AND NOT I_BagArrive[mySelLine] AND NOT Std.HaltSysZone[myZone]) THEN
		D[900 + mySeq] = 5
	ENDIF
	IF Request.IC[mySelLine] AND NOT PUPClear[mySelLine] THEN
		Alarm[mySeq].Bag = myOutBag[mySelLine]
		Alarm[mySeq].Name = almBagDataError
	ELSE IF I_BagArrive[mySelLine] THEN
		Alarm[mySeq].Name = almSwitchFault
	ELSE IF NOT BagValid	AND SettledAtSep THEN
		Alarm[mySeq].Name = almBagDataError
	ELSE IF BagValid AND NOT SettledAtSep THEN
		Alarm[mySeq].Name = almSwitchFault
	ELSE IF NOT Std.HaltSysZone[myZone] THEN
	;	Alarm[mySeq].Name = almBagNotReleased
	ENDIF
ENDIF

;Step 5 Release bag to PUP
IF (STEP = 5) THEN
	mySelLine = 2
	myPrevSelLine = mySelLine
	DestValid = (myDest = myRelDest[mySelLine])
	O_Select[mySelLine] = DestValid
	O_OpenSep = (Request.UP[myPUP[mySelLine]] AND DestValid AND BagValid AND PUPClear[mySelLine] AND NOT BagInSep AND NOT I_BagArrive[mySelLine])
	IF I_BagArrive[mySelLine] AND PUPClear[mySelLine] AND BagValid THEN
		Bag[myOutBag[mySelLine]] = Bag[myBag]
		Bag[myBag] = Bag[0]
		D[900 + mySeq] = 1
	ENDIF
	IF NOT PUPClear[mySelLine] THEN
		Alarm[mySeq].Bag = myOutBag[mySelLine]
		Alarm[mySeq].Name = almBagDataError
	ELSE IF NOT BagValid AND SettledAtSep THEN
		Alarm[mySeq].Name = almBagDataError
	ELSE IF BagValid AND NOT SettledAtSep THEN
		Alarm[mySeq].Name = almSwitchFault
	ELSE IF NOT DestValid AND SettledAtSep THEN
		Alarm[mySeq].Name = almDestinationNotValid
	ENDIF
ENDIF
;-----------------------------------
;PLC Outputs - adjust to suit system
;-----------------------------------

ExitSeq:

Y[myIO].Y05 = O_OpenSep
Y[myIO].Y07 = O_Select[2]
Y[myIO].Y08 = O_Select[1]

;Alarms
TimerAlarm.IN 		= NOT PLS AND (Alarm[mySeq].Name > 0)
TimerAlarm.PT 		= Alarm[mySeq].Time
TimerAlarm FUB TON_10ms()
Alarm[mySeq].On 	= TimerAlarm.Q
Alarm[mySeq].ET 	= TimerAlarm.ET
Alarm[mySeq].Zone 	= myZone
END_PROGRAM
```

### Program Logical/Reference/24_pp10 (IEC) - *PP10 Empty trolleys feeding PICU9

#### pp.var
```iecst
VAR RETAIN
	LASTSTEP : UINT;
	PLS : BOOL;
	STEP : UINT;
END_VAR
VAR
	TimerAlarm : TON_10ms;
	mySeq : UINT;
	myIO : UINT;
	I_BagAtSep : ARRAY[0..2] OF BOOL;
	I_LineFull : BOOL;
	O_OpenSep : ARRAY[0..2] OF BOOL;
	O_Select : ARRAY[0..2] OF BOOL;
	SettledAtSep : ARRAY[0..2] OF BOOL;
	SettledAtSepET : ARRAY[0..2] OF UDINT;
	myLine : USINT;
	TrolleyCount : ARRAY[0..2] OF UINT;
	TrolleyBatchSize : UINT;
	n : UINT;
	I_BufferLineFull : ARRAY[0..2] OF BOOL;
	BufferFull : ARRAY[0..2] OF BOOL;
	BufferFullET : ARRAY[0..2] OF UDINT;
	Reset : BOOL;
	ResetPoints : BOOL;
	ResetPointsET : UDINT;
END_VAR
VAR RETAIN
	myPrevLine : UINT;
END_VAR
VAR
	myZone : INT;
	I_BagInSep : ARRAY[0..2] OF BOOL;
	SettledInSep : ARRAY[0..2] OF BOOL;
	SettledInSepET : ARRAY[0..2] OF UDINT;
	BagInSep : ARRAY[0..2] OF BOOL;
END_VAR
```

#### pp.ab
```automation-basic
;--------------------------------------------
;Sequence 0 - XXX0  D[900 + mySeq]
;--------------------------------------------

PROGRAM _INIT
(* init program *)
END_PROGRAM

PROGRAM _CYCLIC

;Inputs
mySeq				= 24	;Sequence number
myIO				= 110
myZone				= 0

TrolleyBatchSize 	= 4

I_BagAtSep[1]			= X[myIO].X01
I_BagAtSep[2]			= X[myIO].X02
I_BagInSep[1]			= X[178].X08
I_BagInSep[2]			= X[myIO].X04
I_LineFull				= X[myIO].X03
I_BufferLineFull[1]		= X[178].X05
I_BufferLineFull[2]		= X[348].X08

O_OpenSep[1]			= FALSE
O_OpenSep[2]			= FALSE
O_Select[1]				= FALSE
O_Select[2]				= FALSE

Alarm[mySeq].Name 	= 0
Alarm[mySeq].Bag	= 10000 + mySeq
Alarm[mySeq].Beacon	= TRUE
Alarm[mySeq].Extra	= 0
Alarm[mySeq].Time	= 3000

;Setup Sequence
STEP = D[900 + mySeq]
;Setup Pulse contact
PLS = (STEP <> LASTSTEP)
LASTSTEP = STEP

;Keep trolley counts inrange
LOOP n = 1 TO 2 DO
	IF (TrolleyCount[n] >$FFFE) THEN
		TrolleyCount[n] = $FFFE
	ENDIF
ENDLOOP

;Sequence
IF (STEP = 0) THEN
	;Disabled
ENDIF

;Step 1 Decide where to take trolley from
TON_10ms(I_BagAtSep[1],200,SettledAtSep[1],SettledAtSepET[1])
TON_10ms(I_BagAtSep[2],200,SettledAtSep[2],SettledAtSepET[2])
TON_10ms(I_BufferLineFull[1],400,BufferFull[1],BufferFullET[1])
TON_10ms(I_BufferLineFull[2],400,BufferFull[2],BufferFullET[2])
TON_10ms(Reset,200,ResetPoints,ResetPointsET)
IF (STEP = 1) THEN
		;Force line choice if line is full
	IF NOT Reset THEN
		IF BufferFull[1] AND NOT BufferFull[2] THEN
			myLine = 1
		ELSE IF BufferFull[2] AND NOT BufferFull[1] THEN
			myLine = 2
		ENDIF
	ENDIF
	IF (myLine = 0) OR (myLine > 2) THEN
		myLine = 1
	ENDIF

	IF (SettledAtSep[myLine] AND (TrolleyCount[myLine] < TrolleyBatchSize) AND NOT I_LineFull AND NOT Reset AND NOT Std.HaltSysZone[myZone]) THEN
		IF (myLine = myPrevLine) THEN
			D[900 +  mySeq] = (myLine + 1)
		ELSE
			Reset = TRUE
		ENDIF
	ELSE IF Reset THEN
		O_Select[myLine] = TRUE
		IF ResetPoints THEN
			myPrevLine = myLine
			D[900 +  mySeq] = (myLine + 1)
		ENDIF
	ELSE IF (TrolleyCount[myLine] >= TrolleyBatchSize) OR NOT I_BagAtSep[myLine] THEN
		TrolleyCount[myLine] = 0
		INC myLine
	ENDIF
ELSE
	Reset = FALSE
ENDIF

;Step 2 Select Line 1
TON_10ms(I_BagInSep[1],150,SettledInSep[1],SettledInSepET[1])
IF (STEP = 2) THEN
	myLine = 1
	IF SettledInSep[myLine] THEN
		BagInSep[myLine] = TRUE
	ENDIF
	O_Select[myLine] = TRUE
	O_OpenSep[myLine] = NOT BagInSep[myLine]
	IF I_LineFull THEN
		INC TrolleyCount[myLine]
		D[900 + mySeq] = 1
	ENDIF
	Alarm[mySeq].Name = almBagNotReleased
ELSE
	BagInSep[1] = FALSE
ENDIF

;Step 3 Select Line 2
TON_10ms(I_BagInSep[2],150,SettledInSep[2],SettledInSepET[2])
IF (STEP = 3) THEN
	myLine = 2
	IF SettledInSep[myLine] THEN
		BagInSep[myLine] = TRUE
	ENDIF
	O_Select[myLine] = TRUE
	O_OpenSep[myLine] = NOT BagInSep[myLine]
	IF I_LineFull THEN
		INC TrolleyCount[myLine]
		D[900 + mySeq] = 1
	ENDIF
	Alarm[mySeq].Name = almBagNotReleased
ELSE
	BagInSep[2] = FALSE
ENDIF

;-----------------------------------
;PLC Outputs - adjust to suit system
;-----------------------------------

Y[myIO].Y05 = O_OpenSep[1]
Y[myIO].Y06 = O_OpenSep[2]
Y[myIO].Y07 = O_Select[1]
Y[myIO].Y08 = O_Select[2]

;Alarms
TimerAlarm.IN 		= NOT PLS AND (Alarm[mySeq].Name > 0)
TimerAlarm.PT 		= Alarm[mySeq].Time
TimerAlarm FUB TON_10ms()
Alarm[mySeq].On 	= TimerAlarm.Q
Alarm[mySeq].ET 	= TimerAlarm.ET
Alarm[mySeq].Zone 	= myZone
END_PROGRAM
```

### Program Logical/Reference/25_pp11 (IEC) - *PP11 Empty trolleys from PUP 4-6

#### pp.ab
```automation-basic
;--------------------------------------------
;Sequence 0 - XXX0  D[900 + mySeq]
;--------------------------------------------

PROGRAM _INIT
(* init program *)
END_PROGRAM

PROGRAM _CYCLIC

;Inputs
mySeq				= 25	;Sequence number
myIO				= 111
myZone	= 0

TrolleyBatchSize 	= 4

I_BagAtSep[1]			= X[myIO].X01
I_BagAtSep[2]			= X[myIO].X02
I_BagInSep[1]			= X[350].X01
I_BagInSep[2]			= X[350].X02
I_LineFull				= X[myIO].X03
I_BufferLineFull[1]		= X[350].X08
I_BufferLineFull[2]		= X[179].X05

O_OpenSep[1]			= FALSE
O_OpenSep[2]			= FALSE
O_Select[1]				= FALSE
O_Select[2]				= FALSE

Alarm[mySeq].Name 	= 0
Alarm[mySeq].Bag	= 10000 + mySeq
Alarm[mySeq].Beacon	= TRUE
Alarm[mySeq].Extra	= 0
Alarm[mySeq].Time	= 3000

;Setup Sequence
STEP = D[900 + mySeq]
;Setup Pulse contact
PLS = (STEP <> LASTSTEP)
LASTSTEP = STEP

;Keep trolley counts inrange
LOOP n = 1 TO 2 DO
	IF (TrolleyCount[n] >$FFFE) THEN
		TrolleyCount[n] = $FFFE
	ENDIF
ENDLOOP

;Sequence
IF (STEP = 0) THEN
	;Disabled
ENDIF

;Step 1 Decide where to take trolley from
TON_10ms(I_BagAtSep[1],200,SettledAtSep[1],SettledAtSepET[1])
TON_10ms(I_BagAtSep[2],200,SettledAtSep[2],SettledAtSepET[2])
TON_10ms(I_BufferLineFull[1],400,BufferFull[1],BufferFullET[1])
TON_10ms(I_BufferLineFull[2],400,BufferFull[2],BufferFullET[2])
TON_10ms(Reset,200,ResetPoints,ResetPointsET)
IF (STEP = 1) THEN
	;Force line choice if line is full
	IF NOT Reset THEN
		IF BufferFull[1] AND NOT BufferFull[2] THEN
			myLine = 1
		ELSE IF BufferFull[2] AND NOT BufferFull[1] THEN
			myLine = 2
		ENDIF
	ENDIF
	IF (myLine = 0) OR (myLine > 2) THEN
		myLine = 1
	ENDIF

	IF (SettledAtSep[myLine] AND (TrolleyCount[myLine] < TrolleyBatchSize) AND NOT I_LineFull AND NOT Reset AND NOT Std.HaltSysZone[myZone]) THEN
		IF (myLine = myPrevLine) THEN
			D[900 +  mySeq] = (myLine + 1)
		ELSE
			Reset = TRUE
		ENDIF
	ELSE IF Reset THEN
		O_Select[myLine] = TRUE
		IF ResetPoints THEN
			myPrevLine = myLine
			D[900 +  mySeq] = (myLine + 1)
		ENDIF
	ELSE IF (TrolleyCount[myLine] >= TrolleyBatchSize) OR NOT I_BagAtSep[myLine] THEN
		TrolleyCount[myLine] = 0
		INC myLine
	ENDIF
ELSE
	Reset = FALSE
ENDIF

;Step 2 Select Line 1
TON_10ms(I_BagInSep[1],150,SettledInSep[1],SettledInSepET[1])
IF (STEP = 2) THEN
	myLine = 1
	IF SettledInSep[myLine] THEN
		BagInSep[myLine] = TRUE
	ENDIF
	O_Select[myLine] = TRUE
	O_OpenSep[myLine] = NOT BagInSep[myLine]
	IF I_LineFull THEN
		INC TrolleyCount[myLine]
		D[900 + mySeq] = 1
	ENDIF
	Alarm[mySeq].Name = almBagNotReleased
ELSE
	BagInSep[1] = FALSE
ENDIF

;Step 3 Select Line 2
TON_10ms(I_BagInSep[2],150,SettledInSep[2],SettledInSepET[2])
IF (STEP = 3) THEN
	myLine = 2
	IF SettledInSep[myLine] THEN
		BagInSep[myLine] = TRUE
	ENDIF
	O_Select[myLine] = TRUE
	O_OpenSep[myLine] = NOT BagInSep[myLine]
	IF I_LineFull THEN
		INC TrolleyCount[myLine]
		D[900 + mySeq] = 1
	ENDIF
	Alarm[mySeq].Name = almBagNotReleased
ELSE
	BagInSep[2] = FALSE
ENDIF

;-----------------------------------
;PLC Outputs - adjust to suit system
;-----------------------------------

Y[myIO].Y05 = O_OpenSep[1]
Y[myIO].Y06 = O_OpenSep[2]
Y[myIO].Y07 = O_Select[1]
Y[myIO].Y08 = O_Select[2]

;Alarms
TimerAlarm.IN 		= NOT PLS AND (Alarm[mySeq].Name > 0)
TimerAlarm.PT 		= Alarm[mySeq].Time
TimerAlarm FUB TON_10ms()
Alarm[mySeq].On 	= TimerAlarm.Q
Alarm[mySeq].ET 	= TimerAlarm.ET
Alarm[mySeq].Zone 	= myZone
END_PROGRAM
```

### Program Logical/Reference/26_pp12 (IEC) - *PP12 Empty trolleys from PUP 1-6

#### pp.ab
```automation-basic
;--------------------------------------------
;Sequence 0 - XXX0  D[900 + mySeq]
;--------------------------------------------

PROGRAM _INIT
(* init program *)
END_PROGRAM

PROGRAM _CYCLIC

;Inputs
mySeq	= 26	;Sequence number
myIO	= 112
myZone	= 2

TrolleyBatchSize 	= 200; time to open stop

I_BagAtSep[1]			= X[myIO].X01
I_BagAtSep[2]			= X[myIO].X02
I_LineFull				= X[myIO].X03
I_BufferLineFull[1]		= X[252].X03
I_BufferLineFull[2]		= X[251].X03

O_OpenSep[1]			= FALSE
O_OpenSep[2]			= FALSE
O_Select[1]				= FALSE
O_Select[2]				= FALSE

Alarm[mySeq].Name 	= 0
Alarm[mySeq].Bag	= 10000 + mySeq
Alarm[mySeq].Beacon	= TRUE
Alarm[mySeq].Extra	= 0
Alarm[mySeq].Time	= 3000

;Setup Sequence
STEP = D[900 + mySeq]
;Setup Pulse contact
PLS = (STEP <> LASTSTEP)
LASTSTEP = STEP

IF (STEP < 2) THEN
	BatchRecieved = FALSE
ENDIF
;Sequence
IF (STEP = 0) THEN
	;Disabled
ENDIF

;Step 1 Decide where to take trolley from
TON_10ms(I_BagAtSep[1],250,SettledAtSep[1],SettledAtSepET[1])
TON_10ms(I_BagAtSep[2],250,SettledAtSep[2],SettledAtSepET[2])
TON_10ms(I_BufferLineFull[1],400,BufferFull[1],BufferFullET[1])
TON_10ms(I_BufferLineFull[2],400,BufferFull[2],BufferFullET[2])
TON_10ms((STEP > 1),TrolleyBatchSize,CloseStop,CloseStopET)
IF (STEP = 1) THEN
	IF (NOT I_LineFull AND NOT Std.HaltSysZone[myZone]) THEN
		INC myLine
		IF (myLine < 1) OR (myLine > 2) THEN
			myLine = 1
		ENDIF
		IF SettledAtSep[myLine] THEN
			D[900 + mySeq] = 1 + myLine
		ENDIF
	ENDIF
ENDIF

;Step 2 Select Line 1
TON_10ms(BatchRecieved,(TrolleyBatchSize + 200),WholeBatchRecieved,WholeBatchRecievedET)
IF (STEP = 2) THEN
	myLine = 1
	O_Select[myLine] = TRUE
	O_OpenSep[myLine] = NOT CloseStop
	IF I_LineFull AND CloseStop THEN
		BatchRecieved = TRUE
	ENDIF
	IF WholeBatchRecieved THEN
		D[900 + mySeq] = 1
	ENDIF
	Alarm[mySeq].Name = almBagNotReleased
ENDIF

;Step 3 Select Line 2
IF (STEP = 3) THEN
	myLine = 2
	O_Select[myLine] = TRUE
	O_OpenSep[myLine] = NOT CloseStop
	IF I_LineFull AND CloseStop THEN
		BatchRecieved = TRUE
	ENDIF
	IF WholeBatchRecieved THEN
		D[900 + mySeq] = 1
	ENDIF
	Alarm[mySeq].Name = almBagNotReleased
ENDIF

;-----------------------------------
;PLC Outputs - adjust to suit system
;-----------------------------------

Y[myIO].Y05 = O_OpenSep[1]
Y[myIO].Y06 = O_OpenSep[2]
Y[myIO].Y07 = O_Select[1]
Y[myIO].Y08 = O_Select[2]

;Alarms
TimerAlarm.IN 		= NOT PLS AND (Alarm[mySeq].Name > 0)
TimerAlarm.PT 		= Alarm[mySeq].Time
TimerAlarm FUB TON_10ms()
Alarm[mySeq].On 	= TimerAlarm.Q
Alarm[mySeq].ET 	= TimerAlarm.ET
Alarm[mySeq].Zone 	= myZone
END_PROGRAM
```

### Program Logical/Reference/27_pp13 (IEC) - *PP13 Empty trolleys to PICD13 + PP14

#### pp.ab
```automation-basic
;--------------------------------------------
;Sequence 0 - XXX0  D[900 + mySeq]
;--------------------------------------------

PROGRAM _INIT
(* init program *)
END_PROGRAM

PROGRAM _CYCLIC

;Inputs
mySeq				= 27	;Sequence number
myIO				= 113
myZone				= 3
OpenStopTime		= 100

I_BagAtSep			= X[myIO].X01
I_LineFull[1]		= X[myIO].X03
I_LineFull[2]		= X[myIO].X04
I_BufferLineEmpty[1] = 	(NOT X[183].X03 AND NOT Y[183].Y06)
I_BufferLineEmpty[2] = 	(NOT X[114].X01 AND NOT Y[114].Y05)

;TrolleyBatchSize	= 3

O_OpenSep			= FALSE
O_Select[1]			= FALSE
O_Select[2]			= FALSE

Alarm[mySeq].Name 	= 0
Alarm[mySeq].Bag	= 10000 + mySeq
Alarm[mySeq].Beacon	= TRUE
Alarm[mySeq].Extra	= 0
Alarm[mySeq].Time	= 3000

;Setup Sequence
STEP = D[900 + mySeq]
;Setup Pulse contact
PLS = (STEP <> LASTSTEP)
LASTSTEP = STEP

;Sequence
IF (STEP = 0) THEN
	;Disabled
ENDIF

;Step 1 Decide where to send trolley
TON_10ms(I_BagAtSep,250,SettledAtSep,SettledAtSepET)
TON_10ms(I_BufferLineEmpty[1],200,BufferEmpty[1],BufferEmptyET[1])
TON_10ms(I_BufferLineEmpty[2],200,BufferEmpty[2],BufferEmptyET[2])
TON_10ms((STEP = 1),200,ResetPoints,ResetPointsET)
IF (STEP = 1) THEN
	BagsArrived = FALSE
	IF (SettledAtSep AND NOT Std.HaltSysZone[myZone]) THEN
		IF (myLine < 2) THEN
			INC myLine
		ELSE
			myLine = 1
		ENDIF

		IF NOT I_LineFull[myLine]  THEN
			D[900 +  mySeq] = (myLine + 1)
		ENDIF
	ENDIF
ENDIF

TON_10ms((STEP = 2) OR (STEP = 3),OpenStopTime,OpenStop,OpenStopET)
TON_10ms(BagsArrived,OpenStopTime + 100,BagsReleased,BagsReleasedET)
;Step 2 Select Line 1
IF (STEP = 2) THEN
	myLine = 1
		O_Select[myLine] = TRUE
	O_OpenSep = NOT OpenStop
	IF I_LineFull[myLine] THEN
		BagsArrived = TRUE
	ENDIF
	IF BagsReleased THEN
		D[900 + mySeq] = 1
	ENDIF
	Alarm[mySeq].Name = almBagNotReleased
ENDIF

;Step 3 Select Line 2
IF (STEP = 3) THEN
	myLine = 2
	O_Select[myLine] = TRUE
	O_OpenSep = NOT OpenStop
	IF I_LineFull[myLine] THEN
		BagsArrived = TRUE
	ENDIF
	IF BagsReleased THEN
		D[900 + mySeq] = 1
	ENDIF
	Alarm[mySeq].Name = almBagNotReleased
ENDIF

;-----------------------------------
;PLC Outputs - adjust to suit system
;-----------------------------------

Y[myIO].Y05 = O_OpenSep
Y[myIO].Y07 = O_Select[1]
Y[myIO].Y08 = O_Select[2]

;Alarms
TimerAlarm.IN 		= NOT PLS AND (Alarm[mySeq].Name > 0)
TimerAlarm.PT 		= Alarm[mySeq].Time
TimerAlarm FUB TON_10ms()
Alarm[mySeq].On 	= TimerAlarm.Q
Alarm[mySeq].ET 	= TimerAlarm.ET
Alarm[mySeq].Zone 	= myZone
END_PROGRAM
```

### Program Logical/Reference/28_pp14 (IEC) - *PP14 Empty trolleys to PICD14+ PICD15

#### pp.var
```iecst
VAR RETAIN
	LASTSTEP : UINT;
	PLS : BOOL;
	STEP : UINT;
END_VAR
VAR
	TimerAlarm : TON_10ms;
	mySeq : UINT;
	myIO : UINT;
	I_BagAtBuffer : BOOL;
	I_BagAtSep : BOOL;
	I_LineFull : ARRAY[0..2] OF BOOL;
	O_OpenSep : BOOL;
	O_Select : ARRAY[0..2] OF BOOL;
	n : UINT;
	TrolleyCount : ARRAY[0..2] OF UINT;
	SettledAtSep : BOOL;
	SettledAtSepET : UDINT;
	Reset : BOOL;
	ResetPoints : BOOL;
	ResetPointsET : UDINT;
	myLine : UINT;
	TrolleyBatchSize : UINT;
	myPrevLine : UINT;
	I_BufferLineEmpty : ARRAY[0..2] OF BOOL;
	BufferEmpty : ARRAY[0..2] OF BOOL;
	BufferEmptyET : ARRAY[0..2] OF UDINT;
	myZone : INT;
	BagsArrived : BOOL;
	OpenStopTime : UDINT;
	OpenStop : BOOL;
	OpenStopET : UDINT;
	BagsReleased : BOOL;
	BagsReleasedET : UDINT;
END_VAR
```

### Program Logical/Reference/29_pp17 (IEC) - *PP17 Full bags goings onto PIC1&2

#### pp.var
```iecst
VAR RETAIN
	LASTSTEP : UINT;
	PLS : BOOL;
	STEP : UINT;
END_VAR
VAR
	TimerAlarm : TON_10ms;
	mySeq : UINT;
	myIO : UINT;
	I_BagAtSep : ARRAY[0..3] OF BOOL;
	I_ReleasedSep : ARRAY[0..3] OF BOOL;
	O_SelectLine : ARRAY[0..3] OF BOOL;
	O_SelectDest : ARRAY[0..3] OF BOOL;
	TON_Settled : ARRAY[0..3] OF TON_10ms;
	n : UINT;
	myBag : UINT;
	myBuffBag : ARRAY[0..3] OF UINT;
	LineValid : ARRAY[0..4] OF BOOL;
	myRelLine : ARRAY[0..2] OF UINT;
END_VAR
VAR RETAIN
	CurrentDest : UINT;
	CurrentLine : UINT;
END_VAR
VAR
	myDestBag : UINT;
	LineBatchCount : ARRAY[0..3] OF UINT;
	MaxBatchSize : UINT;
	ResetRequired : BOOL;
	ResetPoints : BOOL;
	ResetPointsET : UDINT;
	PrevDest : UINT;
	PrevLine : UINT;
	O_OpenSep : ARRAY[0..3] OF BOOL;
	Released : BOOL;
	myDestLine : UINT;
	ReleaseValid : BOOL;
	ClearCounts : BOOL;
	LineSearchCount : UINT;
	DestSearchCount : UINT;
	ScanUpdate : BOOL;
	ScanUpdateET : UDINT;
	myZone : INT;
	TON_0penStop : ARRAY[0..3] OF TON_10ms;
	x : INT;
	TON_SettledInSep : ARRAY[0..3] OF TON_10ms;
END_VAR
```

#### pp.ab
```automation-basic
;--------------------------------------------
;Sequence 0 - XXX0  D[900 + mySeq]
;--------------------------------------------

PROGRAM _INIT
(* init program *)
END_PROGRAM

PROGRAM _CYCLIC

;Inputs
mySeq				= 29	;Sequence number
myIO				= 115
myZone				= 3

I_BagAtSep[1]		= X[myIO].X01
I_BagAtSep[2]		= X[myIO].X02
I_BagAtSep[3]		= X[myIO + 1].X01
I_ReleasedSep[1]	= X[myIO].X03
I_ReleasedSep[2]	= X[myIO].X04
I_ReleasedSep[3]	= X[myIO + 1].X03

myBuffBag[1]		= 811
myBuffBag[2]		= 801
myBuffBag[3]		= 821

myRelLine[1]		= 63
myRelLine[2]		= 64

MaxBatchSize 		= 3 ; Max number of bags to send from 1 line with out selecting another..

O_SelectLine[1]		= FALSE
O_SelectLine[2]		= FALSE
O_SelectLine[3]		= FALSE

O_OpenSep[1]		= FALSE
O_OpenSep[2]		= FALSE
O_OpenSep[3]		= FALSE

O_SelectDest[1]		= FALSE
O_SelectDest[2]		= FALSE

Alarm[mySeq].Name 	= 0
Alarm[mySeq].Bag	= 10000 + mySeq
Alarm[mySeq].Beacon	= TRUE
Alarm[mySeq].Extra	= 0
Alarm[mySeq].Time	= 3000

;Setup Sequence
STEP = D[900 + mySeq]
;Setup Pulse contact
PLS = (STEP <> LASTSTEP)
LASTSTEP = STEP

;Sequence
IF (STEP = 0) THEN
	;Disabled
ENDIF

LOOP n = 1 TO 3 DO
	TON_Settled[n].IN = I_BagAtSep[n]
	TON_Settled[n].PT = 150
	TON_Settled[n] FUB TON_10ms()
	myBag = myBuffBag[n]
	LineValid[n] = TON_Settled[n].Q AND (Bag[myBag].Cat > 0) AND NOT I_ReleasedSep[n]
	TON_SettledInSep[n].IN = I_ReleasedSep[n]
	TON_SettledInSep[n].PT = 50
	TON_SettledInSep[n] FUB TON_10ms()

	;Alarms
ENDLOOP
;Step 1 Try to find batch with the same category

TON_10ms((STEP =1),5,ScanUpdate,ScanUpdateET)
IF (STEP = 1) AND ScanUpdate THEN ; Allow short time for trips to settle before looking for next batch
	IF (CurrentDest <= 0) OR (CurrentDest > 2) THEN
		CurrentDest = 1
	ENDIF
	IF (CurrentLine <= 0) OR (CurrentLine > 3) THEN
		CurrentLine = 1
	ENDIF
	IF (PrevLine <= 0) OR (PrevLine > 3) THEN
		PrevLine = 1
	ENDIF
	IF (LineBatchCount[CurrentLine] >= MaxBatchSize) AND LineValid[CurrentLine] AND (DestSearchCount > 2) THEN
		LineBatchCount[CurrentLine] = 0
	ENDIF
	myDestLine = myRelLine[CurrentDest]
		IF Line[myDestLine].Clear AND NOT Line[myDestLine].TripFault AND NOT Std.HaltSysZone[myZone] THEN
		;Search for line with matching cat starting at the currently selected line. Ensure we do not send more than a certain number of bags from 1 line.
		myBag = myBuffBag[CurrentLine]
		myDestBag	= (Line[myDestLine].LastBag - Line[myDestLine].Space)

		IF LineValid[CurrentLine] AND (LineBatchCount[CurrentLine] < MaxBatchSize) THEN ; Check line is valid
			IF (Bag[myBag].Cat = Bag[myDestBag].Cat) THEN ; Match Cats.
				D[900 + mySeq] = 2
			ELSE IF (Bag[Line[myDestLine].FirstBag].Cat = 0) THEN ; Line is empty
				D[900 + mySeq] = 2
			ELSE IF (DestSearchCount > 2) THEN ; No matches send any bag
				D[900 + mySeq] = 2
			ELSE
				INC CurrentLine ; Search next line.
				INC LineSearchCount
				IF LineSearchCount > 3 THEN ; Search all lines if nothing search next buffer.
					LineSearchCount = 0
					INC CurrentDest
					INC DestSearchCount
				ENDIF
			ENDIF
		ELSE
			INC CurrentLine ; Search next line.
			INC LineSearchCount
			IF LineSearchCount > 3 THEN ; Search all lines if nothing search next buffer.
				LineSearchCount = 0
				INC CurrentDest
				INC DestSearchCount
			ENDIF
		ENDIF
	ELSE IF NOT Std.HaltSysZone[myZone] THEN
		INC CurrentDest
	ENDIF
ELSE IF (STEP <> 1) THEN
	DestSearchCount = 0
	LineSearchCount	= 0
ENDIF

;Step 2 Select Points if required
TON_10ms(ResetRequired,200,ResetPoints,ResetPointsET)
IF (STEP = 2) THEN
	IF (CurrentDest > 0) AND (CurrentDest < 3) AND (CurrentLine > 0) AND (CurrentLine < 4) THEN
		ResetRequired = ((CurrentDest <> PrevDest) OR (CurrentLine <> PrevLine))
		O_SelectDest[CurrentDest] = TRUE
		O_SelectLine[CurrentLine] = TRUE
		IF NOT ResetRequired OR ResetPoints THEN
			;Clear All other line batch Counts
			LOOP n = 1 TO 3 DO
				IF (n <> CurrentLine) THEN
					LineBatchCount[n] = 0
				ENDIF
			ENDLOOP
			D[900 + mySeq] = 3
		ENDIF
	ELSE
		D[900 + mySeq]  = 1 ; Invalid line/Dest selection reset seq
	ENDIF
ENDIF

;Step 3 Release trolley

IF (STEP = 3) THEN
	IF (CurrentDest > 0) AND (CurrentDest < 3) AND (CurrentLine > 0) AND (CurrentLine < 4) THEN
		myDestLine = myRelLine[CurrentDest]
		myBag = myBuffBag[CurrentLine]
		myDestBag = Line[myDestLine].LastBag

		ReleaseValid = (Bag[myBag].Cat > 0) AND Line[myDestLine].Clear
		O_SelectDest[CurrentDest] = TRUE
		O_SelectLine[CurrentLine] = TRUE
		O_OpenSep[CurrentLine] =  NOT Released;ReleaseValid AND
		IF TON_SettledInSep[CurrentLine].Q THEN
			Released = TRUE
		ENDIF
		IF Line[myDestLine].Trip THEN
			INC LineBatchCount[CurrentLine]
			PrevDest = CurrentDest
			PrevLine = CurrentLine
			Bag[myDestBag] = Bag[myBag]
			Bag[myBag] = Bag[0]
			D[900 + mySeq] = 1
		ENDIF
		IF (Bag[myBag].Cat = 0)THEN
			Alarm[mySeq].Bag = myBag
			Alarm[mySeq].Name = almBagDataError
		ENDIF
	ELSE
		Alarm[mySeq].Time = 0
		Alarm[mySeq].Name = almGeneralSequence
	ENDIF
ELSE
	Released = FALSE
ENDIF

;ClearBatch Counts

IF ClearCounts THEN
	LOOP n = 1 TO 3 DO
		LineBatchCount[n] = 0
	ENDLOOP
	ClearCounts = FALSE
ENDIF
;-----------------------------------
;PLC Outputs - adjust to suit system
;-----------------------------------

Y[myIO].Y05 =  O_OpenSep[1]
Y[myIO].Y06 =  O_OpenSep[2]
Y[myIO + 1].Y05 = O_OpenSep[3]

Y[myIO].Y07 = O_SelectLine[1]
Y[myIO].Y08 = O_SelectLine[2]
Y[myIO + 1].Y07 = O_SelectLine[3]
Y[myIO + 1].Y08 = O_SelectLine[1] OR O_SelectLine[2]

Y[myIO + 2].Y07 = O_SelectDest[1]
Y[myIO + 2].Y08 = O_SelectDest[2]

;Alarms
TimerAlarm.IN 		= NOT PLS AND (Alarm[mySeq].Name > 0)
TimerAlarm.PT 		= Alarm[mySeq].Time
TimerAlarm FUB TON_10ms()
Alarm[mySeq].On 	= TimerAlarm.Q
Alarm[mySeq].ET 	= TimerAlarm.ET
Alarm[mySeq].Zone 	= myZone
END_PROGRAM
```

### Program Logical/Reference/30_picu1 (IEC) - *PICU1 Incline Up Full bags

#### picu.var
```iecst
VAR
	STEP : UINT;
END_VAR
VAR RETAIN
	PLS : BOOL;
	LASTSTEP : UINT;
END_VAR
VAR
	O_RunMotor : BOOL;
	I_OutgoingFull : BOOL;
	O_OpenSeparator : BOOL;
	ReleasedToIncline : BOOL;
	ReleasedToInclineET : TIME;
	NoBags : BOOL;
	StopInclineET : TIME;
	StopIncline : BOOL;
	I_PaddleInPosition : BOOL;
	BagArriveIncline : BOOL;
	I_ArriveIncline : BOOL;
	TransitWindowClosedET : TIME;
	TransitWindowClosed : BOOL;
	BagReleasedSep : BOOL;
	I_BagAtSep : BOOL;
	I_TrolleyOutAtBott : BOOL;
	I_TrolleyOnIncline : BOOL;
	BagReleased : BOOL;
	mySeq : UINT;
	myIO : UINT;
	myBufferBag : UINT;
	myRelLine : UINT;
	myLine : UINT;
	myLastBag : UINT;
	myFirstBag : UINT;
	myX20IO : UINT;
	I_BagReleasedSep : BOOL;
	TimerAlarm : TON_10ms;
	myRelBag : UINT;
	SettledAtSep : BOOL;
	SettledAtSepET : UDINT;
	myZone : INT;
	OpenSep : BOOL;
	OpenSepET : UDINT;
	SettledInSep : BOOL;
	SettledInSepET : UDINT;
	BagArrived : BOOL;
END_VAR
```

### Program Logical/Reference/33_picd4 (IEC) - *PICD4 Incline Down Full bags

#### picd.var
```iecst
VAR
	STEP : UINT;
END_VAR
VAR RETAIN
	PLS : BOOL;
	LASTSTEP : UINT;
END_VAR
VAR
	O_RunMotor : BOOL;
	I_OutgoingFull : BOOL;
	O_OpenSeparator : BOOL;
	ReleasedToIncline : BOOL;
	ReleasedToInclineET : TIME;
	NoBags : BOOL;
	StopInclineET : TIME;
	StopIncline : BOOL;
	I_PaddleInPosition : BOOL;
	BagArriveIncline : BOOL;
	I_ArriveIncline : BOOL;
	TransitWindowClosedET : TIME;
	TransitWindowClosed : BOOL;
	BagReleasedSep : BOOL;
	I_BagAtSep : BOOL;
	I_TrolleyOutAtBott : BOOL;
	I_TrolleyOnIncline : BOOL;
	BagReleased : BOOL;
	mySeq : UINT;
	myIO : UINT;
	myBufferBag : UINT;
	myRelLine : UINT;
	myLine : UINT;
	myLastBag : UINT;
	myFirstBag : UINT;
	myX20IO : UINT;
	I_BagReleasedSep : BOOL;
	TimerAlarm : TON_10ms;
	myRelBag : UINT;
	myIC : UINT;
	DestValid : BOOL;
	myZone : INT;
	I_BagInSep : BOOL;
	SettledAtSep : BOOL;
	SettledAtSepET : UDINT;
	SettledInSep : BOOL;
	SettledInSepET : UDINT;
	BagArrived : BOOL;
END_VAR
```

### Program Logical/Reference/34_picd5 (IEC, version 1.00.0) - *PICD5 Incline Down Full bags

#### picd.ab
```automation-basic
PROGRAM _CYCLIC

;Sequence 24 - Primary Incline Conveyor 1 D[900 + mySeq]

;Note - Not a real sequence and not shown

;-----------------------------------------
;Revision 1.00 17/04/2007 D.J. First Issue
;-----------------------------------------

mySeq = 34
myIC = 5
myIO = 175
myX20IO	= 33
myBufferBag = 908
myRelLine	= 70
myLine = 85 ; Line used to track bags
myZone	= 1

myLastBag = Line[myLine].LastBag
myFirstBag = Line[myLine].FirstBag
myRelBag = Line[myRelLine].LastBag

I_PaddleInPosition		= X[myIO].X01
I_BagInSep				= X[myIO].X02
I_BagAtSep              = X[myIO].X03
I_ArriveIncline			= X[myIO].X04

O_RunMotor 				= FALSE
O_OpenSeparator			= FALSE
Enable.IC[myIC]			= FALSE

Alarm[mySeq].Name 	= 0
Alarm[mySeq].Bag	= myFirstBag
Alarm[mySeq].Beacon	= TRUE
Alarm[mySeq].Extra	= 0
Alarm[mySeq].Time	= 3000

;Setup Sequence
;-----------------------
STEP = D[900 + mySeq]
;Setup Pulse contact
PLS = (STEP <> LASTSTEP)
LASTSTEP = STEP

;If no bags on the buffers then stop the motor
NoBags = (((Bag[myFirstBag].Cat = 0) OR ((STEP = 1) AND Bag[myBufferBag].Cat > 0))  AND ((STEP = 1) AND I_PaddleInPosition))
IF NoBags THEN
	StopIncline = TRUE
ELSE IF (STEP <> 1) THEN
	StopIncline = FALSE
ENDIF

O_RunMotor = (Line[myRelLine].Clear AND NOT Line[myRelLine].TripFault AND NOT Std.HaltSysZone[myZone] AND (STEP <> 2) AND (STEP <> 0))
IF (STEP = 0) THEN

ENDIF

;Run Incline until paddle in position
TON_10ms(I_BagAtSep,25,SettledAtSep,SettledAtSepET)	;75
IF (STEP = 1) THEN
	IF ((I_PaddleInPosition OR StopIncline) AND O_RunMotor AND SettledAtSep AND (Bag[myLastBag].Cat = 0) AND (Bag[myBufferBag].Cat > 0) AND NOT I_BagInSep) THEN
		D[900 + mySeq] = 2
	ENDIF
	IF I_BagInSep THEN
		Alarm[mySeq].Name = almSwitchFault
	ENDIF
ENDIF

;Release Bag into incline

TON_10ms(I_BagInSep,150,SettledInSep,SettledInSepET)
IF (STEP = 2) THEN
	IF SettledInSep THEN
		BagArrived = TRUE
	ENDIF
	O_OpenSeparator	= (Bag[myLastBag].Cat = 0) AND NOT BagArrived
	IF I_ArriveIncline THEN
		IF ((Bag[myBufferBag].Cat > 0) AND (Bag[myLastBag].Cat = 0)) THEN
			Bag[myLastBag] = Bag[myBufferBag]
			Bag[myBufferBag] = Bag[0]
		ENDIF
		D[900 + mySeq] = 3
	ENDIF
	IF (Bag[myLastBag].Cat > 0) THEN
		Alarm[mySeq].Name = almBagDataError
		Alarm[mySeq].Time = 0
		Alarm[mySeq].Bag = myLastBag
	ELSE
		Alarm[mySeq].Name = almBagNotReleased
		Alarm[mySeq].Bag = myBufferBag
	ENDIF
ELSE
	BagArrived = FALSE
ENDIF

;Check not stpped on paddle
IF (STEP = 3) THEN
	IF NOT I_PaddleInPosition THEN
		D[900 + mySeq] = 1
	ENDIF
ENDIF

;Move data from incline..
IF Line[myRelLine].Trip AND (Bag[myFirstBag].Cat > 0) AND (Bag[myRelBag].Cat = 0)  THEN ; Trip includes debounce
	Bag[myRelBag] = Bag[myFirstBag]
	Bag[myFirstBag] = Bag[0]
ENDIF

;Alarms
TimerAlarm.IN 		= NOT PLS AND (Alarm[mySeq].Name > 0)
TimerAlarm.PT 		= Alarm[mySeq].Time
TimerAlarm FUB TON_10ms()
Alarm[mySeq].On 	= TimerAlarm.Q
Alarm[mySeq].ET 	= TimerAlarm.ET
Alarm[mySeq].Zone 	= myZone
Y[myX20IO].Y03 	= O_RunMotor AND NOT StopIncline
Y[myIO].Y06 	= O_OpenSeparator
END_PROGRAM
```
